C09147=1195.626,20.298,-44.972,-179.612,5.706,148.893
C09148=1195.622,20.548,-44.987,-179.609,5.707,148.893
C09149=1195.617,20.797,-45.002,-179.606,5.707,148.892
C09150=1195.611,21.047,-45.017,-179.604,5.708,148.892
C09151=1195.606,21.296,-45.031,-179.602,5.709,148.891
C09152=1195.602,21.545,-45.046,-179.599,5.709,148.890
C09153=1195.596,21.795,-45.061,-179.596,5.710,148.889
C09154=1195.591,22.045,-45.076,-179.594,5.710,148.889
C09155=1195.586,22.294,-45.091,-179.592,5.711,148.888
C09156=1195.581,22.544,-45.106,-179.589,5.711,148.888
C09157=1195.576,22.793,-45.120,-179.586,5.712,148.887
C09158=1195.571,23.042,-45.135,-179.584,5.713,148.887
C09159=1195.566,23.292,-45.150,-179.581,5.713,148.886
C09160=1195.561,23.542,-45.165,-179.579,5.714,148.885
C09161=1195.556,23.791,-45.180,-179.576,5.714,148.885
C09162=1195.551,24.041,-45.195,-179.574,5.715,148.884
C09163=1195.546,24.290,-45.209,-179.571,5.716,148.883
C09164=1195.541,24.539,-45.224,-179.569,5.716,148.883
C09165=1195.536,24.789,-45.240,-179.566,5.717,148.882
C09166=1195.531,25.039,-45.254,-179.563,5.717,148.881
C09167=1195.526,25.288,-45.269,-179.561,5.718,148.881
C09168=1195.520,25.538,-45.284,-179.558,5.719,148.880
C09169=1195.516,25.787,-45.299,-179.555,5.720,148.880
C09170=1195.510,26.036,-45.315,-179.553,5.720,148.879
C09171=1195.505,26.286,-45.329,-179.551,5.721,148.878
C09172=1195.501,26.536,-45.344,-179.548,5.722,148.878
C09173=1195.496,26.785,-45.360,-179.545,5.722,148.877
C09174=1195.491,27.035,-45.374,-179.543,5.723,148.876
C09175=1195.486,27.284,-45.390,-179.540,5.724,148.876
C09176=1195.481,27.533,-45.405,-179.538,5.724,148.875
C09177=1195.475,27.783,-45.420,-179.535,5.725,148.875
C09178=1195.471,28.032,-45.435,-179.533,5.725,148.874
C09179=1195.465,28.282,-45.450,-179.530,5.726,148.873
C09180=1195.460,28.551,-45.466,-179.528,5.727,148.873
C09181=1195.454,28.820,-45.482,-179.525,5.727,148.872
C09182=1195.449,29.088,-45.499,-179.522,5.728,148.871
C09183=1195.444,29.357,-45.515,-179.519,5.729,148.871
C09184=1195.439,29.606,-45.530,-179.517,5.730,148.870
C09185=1195.434,29.856,-45.546,-179.514,5.730,148.869
C09186=1195.429,30.106,-45.560,-179.512,5.731,148.869
C09187=1195.424,30.355,-45.576,-179.509,5.731,148.868
C09188=1195.419,30.604,-45.591,-179.506,5.732,148.868
C09189=1195.414,30.854,-45.606,-179.504,5.732,148.867
C09190=1195.409,31.104,-45.621,-179.502,5.733,148.866
C09191=1195.403,31.353,-45.636,-179.499,5.734,148.866
C09192=1195.399,31.603,-45.652,-179.496,5.734,148.865
C09193=1195.394,31.852,-45.667,-179.494,5.735,148.865
C09194=1195.389,32.102,-45.683,-179.492,5.736,148.864
C09195=1195.384,32.351,-45.698,-179.489,5.736,148.863
C09196=1195.378,32.601,-45.713,-179.486,5.737,148.863
C09197=1195.374,32.850,-45.728,-179.484,5.738,148.862
C09198=1195.369,33.100,-45.744,-179.481,5.738,148.861
C09199=1195.364,33.349,-45.759,-179.479,5.739,148.861
C09200=1195.359,33.598,-45.774,-179.476,5.740,148.860
C09201=1195.353,33.848,-45.790,-179.473,5.741,148.860
C09202=1195.349,34.097,-45.805,-179.471,5.741,148.859
C09203=1195.344,34.347,-45.821,-179.468,5.742,148.858
C09204=1195.339,34.596,-45.836,-179.466,5.742,148.858
C09205=1195.334,34.845,-45.851,-179.463,5.743,148.857
C09206=1195.328,35.095,-45.866,-179.461,5.744,148.857
C09207=1195.324,35.345,-45.881,-179.458,5.744,148.856
C09208=1195.319,35.595,-45.897,-179.456,5.745,148.855
C09209=1195.313,35.844,-45.913,-179.453,5.746,148.855
C09210=1195.309,36.093,-45.928,-179.451,5.746,148.854
C09211=1195.303,36.343,-45.943,-179.448,5.747,148.853
C09212=1195.299,36.592,-45.959,-179.446,5.748,148.853
C09213=1195.294,36.842,-45.974,-179.443,5.748,148.852
C09214=1195.289,37.091,-45.990,-179.440,5.750,148.852
C09215=1195.283,37.341,-46.005,-179.437,5.750,148.851
C09216=1195.279,37.590,-46.021,-179.435,5.751,148.850
C09217=1195.274,37.840,-46.036,-179.433,5.751,148.850
C09218=1195.268,38.089,-46.052,-179.430,5.752,148.849
C09219=1195.264,38.338,-46.067,-179.428,5.753,148.849
C09220=1195.259,38.588,-46.083,-179.425,5.753,148.848
C09221=1195.254,38.837,-46.099,-179.422,5.754,148.847
C09222=1195.249,39.086,-46.114,-179.420,5.754,148.847
C09223=1195.244,39.336,-46.130,-179.418,5.755,148.846
C09224=1195.239,39.586,-46.146,-179.415,5.756,148.846
C09225=1195.234,39.835,-46.161,-179.412,5.757,148.845
C09226=1195.229,40.084,-46.176,-179.410,5.758,148.844
C09227=1195.224,40.334,-46.192,-179.407,5.759,148.844
C09228=1195.219,40.584,-46.208,-179.404,5.759,148.843
C09229=1195.213,40.833,-46.223,-179.402,5.760,148.842
C09230=1195.209,41.083,-46.239,-179.400,5.761,148.842
C09231=1195.204,41.332,-46.255,-179.397,5.761,148.841
C09232=1195.199,41.581,-46.271,-179.394,5.762,148.841
C09233=1195.194,41.830,-46.286,-179.392,5.762,148.840
C09234=1195.189,42.081,-46.302,-179.389,5.763,148.839
C09235=1195.184,42.330,-46.317,-179.386,5.764,148.839
C09236=1195.179,42.578,-46.334,-179.384,5.765,148.838
C09237=1195.174,42.829,-46.349,-179.381,5.766,148.838
C09238=1195.169,43.078,-46.365,-179.379,5.766,148.837
C09239=1195.163,43.327,-46.381,-179.376,5.767,148.836
C09240=1195.159,43.577,-46.397,-179.374,5.768,148.836
C09241=1195.154,43.826,-46.412,-179.371,5.768,148.835
C09242=1195.150,44.076,-46.428,-179.369,5.769,148.835
C09243=1195.144,44.325,-46.444,-179.366,5.770,148.834
C09244=1195.139,44.575,-46.459,-179.363,5.771,148.833
C09245=1195.134,44.824,-46.476,-179.361,5.771,148.833
C09246=1195.129,45.074,-46.492,-179.358,5.772,148.832
C09247=1195.124,45.323,-46.507,-179.356,5.773,148.832
C09248=1195.120,45.572,-46.523,-179.353,5.773,148.831
C09249=1195.114,45.822,-46.539,-179.351,5.774,148.830
C09250=1195.110,46.072,-46.555,-179.349,5.775,148.830
C09251=1195.105,46.321,-46.571,-179.345,5.776,148.829
C09252=1195.099,46.570,-46.587,-179.343,5.777,148.829
C09253=1195.094,46.820,-46.603,-179.341,5.778,148.828
C09254=1195.089,47.069,-46.619,-179.338,5.778,148.827
C09255=1195.084,47.319,-46.635,-179.335,5.779,148.827
C09256=1195.079,47.568,-46.651,-179.333,5.779,148.826
C09257=1195.074,47.817,-46.667,-179.330,5.780,148.826
C09258=1195.069,48.067,-46.683,-179.327,5.781,148.825
C09259=1195.065,48.316,-46.698,-179.325,5.782,148.824
C09260=1195.060,48.566,-46.715,-179.322,5.783,148.824
C09261=1195.055,48.815,-46.730,-179.320,5.783,148.823
C09262=1195.050,49.065,-46.747,-179.317,5.784,148.823
C09263=1195.045,49.314,-46.762,-179.315,5.785,148.822
C09264=1195.040,49.563,-46.779,-179.312,5.785,148.821
C09265=1195.035,49.813,-46.795,-179.309,5.787,148.821
C09266=1195.030,50.062,-46.811,-179.307,5.787,148.820
C09267=1195.025,50.312,-46.827,-179.304,5.788,148.820
C09268=1195.020,50.561,-46.842,-179.302,5.789,148.819
C09269=1195.015,50.811,-46.859,-179.299,5.789,148.818
C09270=1195.010,51.060,-46.875,-179.297,5.790,148.818
C09271=1195.005,51.310,-46.891,-179.294,5.790,148.817
C09272=1195.000,51.559,-46.907,-179.291,5.792,148.817
C09273=1194.996,51.809,-46.924,-179.289,5.793,148.816
C09274=1194.990,52.057,-46.940,-179.286,5.793,148.815
C09275=1194.986,52.307,-46.956,-179.284,5.794,148.815
C09276=1194.981,52.556,-46.972,-179.282,5.795,148.814
C09277=1194.976,52.806,-46.988,-179.279,5.795,148.814
C09278=1194.971,53.055,-47.004,-179.276,5.797,148.813
C09279=1194.965,53.306,-47.021,-179.274,5.797,148.813
C09280=1194.960,53.554,-47.037,-179.271,5.798,148.812
C09281=1194.955,53.804,-47.053,-179.268,5.799,148.811
C09282=1194.950,54.053,-47.070,-179.266,5.799,148.811
C09283=1194.946,54.303,-47.086,-179.263,5.800,148.810
C09284=1194.940,54.571,-47.103,-179.260,5.801,148.809
C09285=1194.935,54.839,-47.121,-179.258,5.802,148.809
C09286=1194.930,55.108,-47.138,-179.254,5.803,148.808
C09287=1194.924,55.377,-47.156,-179.252,5.804,148.808
C09288=1194.919,55.626,-47.173,-179.250,5.805,148.807
C09289=1194.914,55.875,-47.189,-179.247,5.805,148.806
C09290=1194.909,56.125,-47.205,-179.245,5.806,148.806
C09291=1194.904,56.374,-47.221,-179.242,5.807,148.805
C09292=1194.900,56.624,-47.238,-179.239,5.808,148.805
C09293=1194.894,56.873,-47.253,-179.237,5.809,148.804
C09294=1194.889,57.123,-47.271,-179.234,5.809,148.803
C09295=1194.885,57.372,-47.287,-179.232,5.810,148.803
C09296=1194.880,57.621,-47.304,-179.229,5.812,148.802
C09297=1194.875,57.871,-47.320,-179.226,5.812,148.802
C09298=1194.870,58.120,-47.336,-179.224,5.813,148.801
C09299=1194.865,58.370,-47.353,-179.221,5.814,148.801
C09300=1194.859,58.619,-47.370,-179.219,5.814,148.800
C09301=1194.855,58.869,-47.385,-179.216,5.815,148.799
C09302=1194.850,59.118,-47.402,-179.213,5.816,148.799
C09303=1194.845,59.367,-47.418,-179.211,5.817,148.798
C09304=1194.840,59.617,-47.436,-179.208,5.817,148.798
C09305=1194.835,59.866,-47.452,-179.206,5.818,148.797
C09306=1194.830,60.116,-47.468,-179.203,5.820,148.796
C09307=1194.826,60.365,-47.485,-179.200,5.820,148.796
C09308=1194.820,60.614,-47.502,-179.198,5.821,148.795
C09309=1194.815,60.864,-47.518,-179.195,5.822,148.795
C09310=1194.811,61.113,-47.535,-179.193,5.822,148.794
C09311=1194.806,61.362,-47.551,-179.190,5.824,148.794
C09312=1194.800,61.612,-47.568,-179.187,5.824,148.793
C09313=1194.796,61.862,-47.584,-179.185,5.825,148.792
C09314=1194.791,62.111,-47.601,-179.183,5.826,148.792
C09315=1194.785,62.360,-47.618,-179.179,5.827,148.791
C09316=1194.781,62.610,-47.635,-179.177,5.828,148.791
C09317=1194.776,62.859,-47.651,-179.175,5.829,148.790
C09318=1194.771,63.108,-47.668,-179.172,5.829,148.789
C09319=1194.766,63.358,-47.685,-179.170,5.830,148.789
C09320=1194.761,63.607,-47.701,-179.167,5.831,148.788
C09321=1194.757,63.856,-47.718,-179.164,5.832,148.788
C09322=1194.751,64.106,-47.735,-179.162,5.833,148.787
C09323=1194.746,64.355,-47.751,-179.159,5.833,148.787
C09324=1194.742,64.604,-47.768,-179.157,5.835,148.786
C09325=1194.737,64.854,-47.785,-179.154,5.836,148.785
C09326=1194.731,65.103,-47.802,-179.151,5.836,148.785
C09327=1194.726,65.353,-47.819,-179.149,5.837,148.784
C09328=1194.722,65.602,-47.836,-179.146,5.838,148.784
C09329=1194.717,65.851,-47.852,-179.143,5.839,148.783
C09330=1194.711,66.101,-47.869,-179.141,5.840,148.783
C09331=1194.707,66.350,-47.886,-179.138,5.840,148.782
C09332=1194.703,66.600,-47.902,-179.135,5.842,148.781
C09333=1194.697,66.849,-47.919,-179.133,5.843,148.781
C09334=1194.692,67.098,-47.936,-179.131,5.843,148.780
C09335=1194.687,67.348,-47.953,-179.128,5.844,148.780
C09336=1194.683,67.598,-47.970,-179.125,5.846,148.779
C09337=1194.677,67.847,-47.987,-179.123,5.846,148.778
C09338=1194.672,68.096,-48.004,-179.120,5.847,148.778
C09339=1194.668,68.346,-48.020,-179.118,5.848,148.777
C09340=1194.663,68.595,-48.038,-179.115,5.849,148.777
C09341=1194.658,68.844,-48.055,-179.112,5.850,148.776
C09342=1194.653,69.093,-48.072,-179.110,5.850,148.776
C09343=1194.648,69.343,-48.088,-179.108,5.851,148.775
C09344=1194.643,69.593,-48.106,-179.104,5.853,148.774
C09345=1194.638,69.841,-48.122,-179.102,5.853,148.774
C09346=1194.633,70.091,-48.140,-179.100,5.854,148.773
C09347=1194.628,70.340,-48.157,-179.097,5.855,148.773
C09348=1194.623,70.590,-48.174,-179.094,5.856,148.772
C09349=1194.619,70.839,-48.191,-179.092,5.857,148.772
C09350=1194.613,71.088,-48.207,-179.089,5.857,148.771
C09351=1194.609,71.337,-48.225,-179.087,5.858,148.771
C09352=1194.603,71.587,-48.242,-179.084,5.860,148.770
C09353=1194.599,71.837,-48.259,-179.082,5.861,148.769
C09354=1194.594,72.086,-48.276,-179.079,5.861,148.769
C09355=1194.589,72.335,-48.293,-179.076,5.862,148.768
C09356=1194.584,72.584,-48.310,-179.074,5.863,148.768
C09357=1194.579,72.834,-48.328,-179.071,5.864,148.767
C09358=1194.574,73.084,-48.344,-179.069,5.865,148.767
C09359=1194.569,73.333,-48.362,-179.066,5.866,148.766
C09360=1194.565,73.582,-48.379,-179.063,5.867,148.765
C09361=1194.559,73.831,-48.396,-179.061,5.868,148.765
C09362=1194.555,74.080,-48.413,-179.058,5.869,148.764
C09363=1194.549,74.330,-48.430,-179.055,5.870,148.764
C09364=1194.544,74.580,-48.448,-179.053,5.870,148.763
C09365=1194.540,74.829,-48.465,-179.050,5.871,148.762
C09366=1194.535,75.079,-48.482,-179.047,5.873,148.762
C09367=1194.530,75.328,-48.499,-179.045,5.873,148.761
C09368=1194.525,75.576,-48.517,-179.043,5.874,148.761
C09369=1194.520,75.826,-48.534,-179.040,5.876,148.760
C09370=1194.515,76.075,-48.551,-179.037,5.876,148.760
C09371=1194.510,76.325,-48.569,-179.035,5.877,148.759
C09372=1194.505,76.575,-48.586,-179.032,5.878,148.759
C09373=1194.501,76.824,-48.603,-179.029,5.879,148.758
C09374=1194.496,77.073,-48.621,-179.027,5.880,148.758
C09375=1194.491,77.323,-48.638,-179.025,5.881,148.757
C09376=1194.486,77.572,-48.655,-179.021,5.882,148.756
C09377=1194.481,77.821,-48.673,-179.019,5.883,148.756
C09378=1194.476,78.070,-48.690,-179.017,5.884,148.755
C09379=1194.471,78.319,-48.707,-179.013,5.885,148.755
C09380=1194.466,78.569,-48.725,-179.011,5.886,148.754
C09381=1194.461,78.818,-48.743,-179.009,5.886,148.754
C09382=1194.456,79.068,-48.760,-179.006,5.888,148.753
C09383=1194.452,79.317,-48.777,-179.003,5.889,148.753
C09384=1194.447,79.567,-48.795,-179.001,5.889,148.752
C09385=1194.442,79.816,-48.813,-178.998,5.891,148.751
C09386=1194.436,80.066,-48.830,-178.995,5.892,148.751
C09387=1194.432,80.314,-48.847,-178.993,5.892,148.750
C09388=1194.427,80.583,-48.866,-178.990,5.894,148.750
C09389=1194.421,80.851,-48.885,-178.987,5.894,148.749
C09390=1194.416,81.120,-48.904,-178.984,5.896,148.748
C09391=1194.411,81.388,-48.923,-178.982,5.897,148.748
C09392=1194.406,81.638,-48.940,-178.979,5.898,148.747
C09393=1194.401,81.887,-48.958,-178.977,5.899,148.747
C09394=1194.396,82.136,-48.975,-178.974,5.899,148.746
C09395=1194.391,82.386,-48.993,-178.971,5.901,148.746
C09396=1194.386,82.635,-49.011,-178.969,5.902,148.745
C09397=1194.381,82.885,-49.028,-178.966,5.902,148.745
C09398=1194.377,83.133,-49.046,-178.963,5.904,148.744
C09399=1194.372,83.383,-49.064,-178.961,5.905,148.743
C09400=1194.367,83.632,-49.081,-178.959,5.906,148.743
C09401=1194.362,83.882,-49.099,-178.955,5.907,148.742
C09402=1194.357,84.131,-49.117,-178.953,5.908,148.742
C09403=1194.352,84.380,-49.135,-178.951,5.908,148.741
C09404=1194.347,84.630,-49.152,-178.948,5.910,148.741
C09405=1194.343,84.879,-49.169,-178.945,5.911,148.740
C09406=1194.338,85.128,-49.187,-178.943,5.911,148.740
C09407=1194.333,85.378,-49.205,-178.940,5.913,148.739
C09408=1194.328,85.627,-49.223,-178.937,5.914,148.739
C09409=1194.323,85.876,-49.241,-178.935,5.914,148.738
C09410=1194.318,86.125,-49.259,-178.932,5.916,148.737
C09411=1194.313,86.374,-49.277,-178.930,5.917,148.737
C09412=1194.308,86.624,-49.294,-178.927,5.918,148.736
C09413=1194.303,86.873,-49.312,-178.925,5.919,148.736
C09414=1194.299,87.122,-49.329,-178.922,5.920,148.735
C09415=1194.294,87.371,-49.347,-178.919,5.921,148.735
C09416=1194.289,87.621,-49.366,-178.917,5.922,148.734
C09417=1194.284,87.871,-49.383,-178.914,5.922,148.734
C09418=1194.279,88.120,-49.401,-178.911,5.924,148.733
C09419=1194.274,88.369,-49.419,-178.909,5.925,148.733
C09420=1194.269,88.619,-49.437,-178.906,5.926,148.732
C09421=1194.265,88.868,-49.455,-178.903,5.927,148.731
C09422=1194.260,89.117,-49.473,-178.901,5.928,148.731
C09423=1194.255,89.366,-49.491,-178.898,5.929,148.730
C09424=1194.250,89.615,-49.509,-178.896,5.930,148.730
C09425=1194.245,89.864,-49.527,-178.893,5.931,148.729
C09426=1194.240,90.115,-49.544,-178.891,5.933,148.729
C09427=1194.235,90.364,-49.562,-178.888,5.933,148.728
C09428=1194.230,90.613,-49.580,-178.885,5.935,148.728
C09429=1194.226,90.862,-49.598,-178.883,5.935,148.727
C09430=1194.221,91.112,-49.616,-178.880,5.936,148.727
C09431=1194.216,91.361,-49.634,-178.877,5.938,148.726
C09432=1194.211,91.610,-49.652,-178.875,5.939,148.726
C09433=1194.206,91.859,-49.670,-178.872,5.940,148.725
C09434=1194.202,92.109,-49.688,-178.870,5.941,148.725
C09435=1194.196,92.358,-49.707,-178.867,5.941,148.724
C09436=1194.191,92.608,-49.725,-178.864,5.943,148.723
C09437=1194.186,92.857,-49.743,-178.862,5.944,148.723
C09438=1194.181,93.106,-49.761,-178.859,5.945,148.722
C09439=1194.176,93.355,-49.779,-178.857,5.946,148.722
C09440=1194.172,93.605,-49.797,-178.854,5.947,148.721
C09441=1194.167,93.854,-49.815,-178.851,5.948,148.721
C09442=1194.162,94.103,-49.834,-178.849,5.949,148.720
C09443=1194.158,94.352,-49.852,-178.846,5.951,148.720
C09444=1194.153,94.601,-49.870,-178.843,5.951,148.719
C09445=1194.148,94.851,-49.889,-178.841,5.952,148.719
C09446=1194.143,95.100,-49.907,-178.838,5.954,148.718
C09447=1194.138,95.350,-49.925,-178.836,5.954,148.718
C09448=1194.133,95.599,-49.943,-178.833,5.956,148.717
C09449=1194.128,95.848,-49.961,-178.830,5.957,148.717
C09450=1194.124,96.098,-49.979,-178.827,5.958,148.716
C09451=1194.119,96.346,-49.998,-178.825,5.959,148.715
C09452=1194.113,96.596,-50.016,-178.822,5.960,148.715
C09453=1194.108,96.845,-50.034,-178.820,5.961,148.714
C09454=1194.104,97.095,-50.053,-178.817,5.962,148.714
C09455=1194.099,97.344,-50.071,-178.814,5.964,148.713
C09456=1194.095,97.593,-50.089,-178.812,5.965,148.713
C09457=1194.089,97.842,-50.108,-178.810,5.965,148.712
C09458=1194.084,98.091,-50.126,-178.807,5.967,148.712
C09459=1194.080,98.341,-50.144,-178.804,5.967,148.711
C09460=1194.075,98.590,-50.163,-178.802,5.969,148.711
C09461=1194.069,98.839,-50.182,-178.799,5.970,148.710
C09462=1194.065,99.089,-50.200,-178.796,5.972,148.710
C09463=1194.060,99.338,-50.218,-178.794,5.972,148.709
C09464=1194.056,99.587,-50.237,-178.791,5.974,148.709
C09465=1194.050,99.836,-50.255,-178.788,5.974,148.708
C09466=1194.046,100.086,-50.274,-178.786,5.975,148.708
C09467=1194.041,100.335,-50.292,-178.783,5.977,148.707
C09468=1194.036,100.584,-50.310,-178.781,5.978,148.707
C09469=1194.031,100.834,-50.329,-178.778,5.979,148.706
C09470=1194.026,101.083,-50.348,-178.776,5.980,148.706
C09471=1194.022,101.332,-50.366,-178.772,5.981,148.705
C09472=1194.016,101.581,-50.384,-178.770,5.982,148.704
C09473=1194.012,101.831,-50.403,-178.767,5.984,148.704
C09474=1194.007,102.080,-50.421,-178.765,5.985,148.703
C09475=1194.001,102.329,-50.440,-178.762,5.986,148.703
C09476=1193.997,102.579,-50.459,-178.760,5.987,148.702
C09477=1193.992,102.828,-50.477,-178.758,5.988,148.702
C09478=1193.987,103.077,-50.496,-178.754,5.989,148.701
C09479=1193.983,103.327,-50.515,-178.752,5.990,148.701
C09480=1193.978,103.575,-50.533,-178.749,5.992,148.700
C09481=1193.973,103.825,-50.552,-178.747,5.992,148.700
C09482=1193.968,104.074,-50.570,-178.744,5.994,148.699
C09483=1193.964,104.323,-50.589,-178.742,5.995,148.699
C09484=1193.959,104.573,-50.608,-178.738,5.996,148.698
C09485=1193.954,104.822,-50.627,-178.736,5.997,148.698
C09486=1193.948,105.071,-50.645,-178.733,5.998,148.697
C09487=1193.944,105.320,-50.664,-178.731,5.999,148.697
C09488=1193.939,105.570,-50.682,-178.728,6.001,148.696
C09489=1193.934,105.819,-50.702,-178.726,6.002,148.696
C09490=1193.930,106.068,-50.721,-178.723,6.003,148.695
C09491=1193.924,106.317,-50.739,-178.720,6.004,148.695
C09492=1193.920,106.586,-50.760,-178.718,6.006,148.694
C09493=1193.914,106.854,-50.780,-178.715,6.006,148.694
C09494=1193.909,107.123,-50.800,-178.712,6.008,148.693
C09495=1193.904,107.391,-50.820,-178.709,6.009,148.693
C09496=1193.899,107.640,-50.839,-178.706,6.010,148.692
C09497=1193.894,107.889,-50.857,-178.704,6.012,148.691
C09498=1193.889,108.139,-50.877,-178.701,6.012,148.691
C09499=1193.884,108.388,-50.895,-178.698,6.014,148.690
C09500=1193.880,108.637,-50.915,-178.696,6.015,148.690
C09501=1193.875,108.886,-50.933,-178.693,6.016,148.689
C09502=1193.870,109.136,-50.952,-178.691,6.017,148.689
C09503=1193.865,109.385,-50.971,-178.688,6.019,148.688
C09504=1193.861,109.634,-50.991,-178.686,6.020,148.688
C09505=1193.856,109.883,-51.009,-178.682,6.021,148.687
C09506=1193.850,110.132,-51.028,-178.680,6.022,148.687
C09507=1193.846,110.382,-51.047,-178.678,6.024,148.686
C09508=1193.841,110.631,-51.066,-178.675,6.024,148.686
C09509=1193.836,110.881,-51.085,-178.672,6.026,148.685
C09510=1193.831,111.129,-51.104,-178.670,6.027,148.685
C09511=1193.827,111.379,-51.124,-178.667,6.028,148.684
C09512=1193.822,111.628,-51.142,-178.665,6.029,148.684
C09513=1193.817,111.878,-51.161,-178.662,6.031,148.683
C09514=1193.812,112.126,-51.180,-178.660,6.032,148.683
C09515=1193.808,112.376,-51.200,-178.656,6.033,148.682
C09516=1193.802,112.625,-51.219,-178.654,6.034,148.682
C09517=1193.798,112.874,-51.237,-178.651,6.035,148.681
C09518=1193.793,113.123,-51.257,-178.648,6.037,148.681
C09519=1193.788,113.373,-51.276,-178.646,6.038,148.680
C09520=1193.783,113.621,-51.295,-178.643,6.040,148.680
C09521=1193.779,113.871,-51.315,-178.641,6.040,148.679
C09522=1193.774,114.119,-51.333,-178.638,6.042,148.679
C09523=1193.769,114.370,-51.352,-178.636,6.043,148.678
C09524=1193.764,114.619,-51.371,-178.633,6.045,148.678
C09525=1193.760,114.868,-51.391,-178.630,6.045,148.677
C09526=1193.754,115.117,-51.410,-178.628,6.047,148.677
C09527=1193.750,115.366,-51.429,-178.625,6.047,148.676
C09528=1193.745,115.616,-51.449,-178.622,6.049,148.676
C09529=1193.740,115.864,-51.468,-178.620,6.050,148.675
C09530=1193.735,116.114,-51.488,-178.617,6.052,148.675
C09531=1193.730,116.363,-51.507,-178.614,6.053,148.674
C09532=1193.726,116.612,-51.526,-178.612,6.054,148.674
C09533=1193.721,116.861,-51.545,-178.609,6.056,148.673
C09534=1193.716,117.110,-51.565,-178.607,6.057,148.673
C09535=1193.711,117.360,-51.584,-178.604,6.058,148.672
C09536=1193.707,117.609,-51.603,-178.602,6.059,148.672
C09537=1193.702,117.858,-51.623,-178.599,6.061,148.672
C09538=1193.697,118.107,-51.642,-178.596,6.061,148.671
C09539=1193.692,118.357,-51.662,-178.594,6.063,148.671
C09540=1193.688,118.606,-51.681,-178.590,6.064,148.670
C09541=1193.683,118.855,-51.700,-178.588,6.065,148.669
C09542=1193.678,119.104,-51.720,-178.586,6.067,148.669
C09543=1193.672,119.353,-51.739,-178.583,6.068,148.668
C09544=1193.668,119.603,-51.759,-178.580,6.069,148.668
C09545=1193.664,119.852,-51.778,-178.578,6.070,148.668
C09546=1193.658,120.101,-51.797,-178.575,6.072,148.667
C09547=1193.654,120.350,-51.817,-178.573,6.073,148.667
C09548=1193.649,120.600,-51.836,-178.570,6.074,148.666
C09549=1193.643,120.849,-51.856,-178.567,6.076,148.666
C09550=1193.639,121.098,-51.875,-178.565,6.077,148.665
C09551=1193.634,121.346,-51.895,-178.562,6.078,148.665
C09552=1193.630,121.596,-51.914,-178.559,6.079,148.664
C09553=1193.625,121.846,-51.934,-178.557,6.081,148.664
C09554=1193.620,122.094,-51.953,-178.554,6.082,148.663
C09555=1193.615,122.344,-51.973,-178.551,6.083,148.663
C09556=1193.610,122.594,-51.993,-178.549,6.085,148.662
C09557=1193.606,122.841,-52.012,-178.546,6.086,148.662
C09558=1193.601,123.091,-52.032,-178.543,6.087,148.661
C09559=1193.596,123.341,-52.051,-178.541,6.088,148.661
C09560=1193.592,123.590,-52.071,-178.538,6.090,148.660
C09561=1193.587,123.838,-52.091,-178.535,6.091,148.660
C09562=1193.582,124.088,-52.111,-178.533,6.092,148.659
C09563=1193.577,124.338,-52.130,-178.530,6.094,148.659
C09564=1193.572,124.586,-52.150,-178.528,6.095,148.658
C09565=1193.567,124.835,-52.170,-178.525,6.096,148.658
C09566=1193.563,125.085,-52.190,-178.522,6.098,148.657
C09567=1193.558,125.335,-52.209,-178.520,6.099,148.657
C09568=1193.553,125.583,-52.229,-178.517,6.101,148.657
C09569=1193.548,125.832,-52.249,-178.515,6.101,148.656
C09570=1193.543,126.082,-52.269,-178.512,6.103,148.656
C09571=1193.539,126.331,-52.289,-178.509,6.105,148.655
C09572=1193.534,126.580,-52.308,-178.507,6.105,148.655
C09573=1193.529,126.829,-52.328,-178.504,6.107,148.654
C09574=1193.524,127.078,-52.348,-178.501,6.109,148.654
C09575=1193.520,127.328,-52.368,-178.499,6.109,148.653
C09576=1193.514,127.577,-52.387,-178.496,6.111,148.653
C09577=1193.510,127.826,-52.408,-178.494,6.112,148.652
C09578=1193.505,128.075,-52.427,-178.491,6.114,148.652
C09579=1193.501,128.324,-52.448,-178.488,6.115,148.651
C09580=1193.495,128.573,-52.467,-178.486,6.116,148.651
C09581=1193.491,128.822,-52.487,-178.483,6.118,148.650
C09582=1193.486,129.072,-52.507,-178.480,6.119,148.650
C09583=1193.482,129.320,-52.527,-178.478,6.120,148.650
C09584=1193.477,129.570,-52.547,-178.475,6.122,148.649
C09585=1193.472,129.819,-52.566,-178.473,6.123,148.648
C09586=1193.467,130.068,-52.587,-178.470,6.124,148.648
C09587=1193.462,130.317,-52.606,-178.467,6.126,148.647
C09588=1193.458,130.566,-52.627,-178.465,6.127,148.647
C09589=1193.453,130.816,-52.646,-178.462,6.129,148.647
C09590=1193.448,131.064,-52.666,-178.459,6.130,148.646
C09591=1193.443,131.313,-52.687,-178.457,6.131,148.646
C09592=1193.438,131.563,-52.707,-178.454,6.133,148.645
C09593=1193.434,131.812,-52.727,-178.451,6.134,148.645
C09594=1193.429,132.062,-52.747,-178.449,6.135,148.644
C09595=1193.425,132.310,-52.767,-178.446,6.137,148.644
C09596=1193.419,132.579,-52.789,-178.443,6.139,148.643
C09597=1193.414,132.847,-52.811,-178.440,6.140,148.643
C09598=1193.409,133.116,-52.833,-178.438,6.141,148.642
C09599=1193.404,133.385,-52.854,-178.435,6.142,148.642
C09600=1193.399,133.634,-52.874,-178.432,6.144,148.641
C09601=1193.394,133.883,-52.895,-178.429,6.146,148.641
C09602=1193.389,134.133,-52.915,-178.427,6.146,148.640
C09603=1193.384,134.381,-52.935,-178.424,6.148,148.640
C09604=1193.380,134.630,-52.955,-178.422,6.150,148.640
C09605=1193.375,134.880,-52.975,-178.419,6.151,148.639
C09606=1193.370,135.129,-52.996,-178.416,6.152,148.639
C09607=1193.366,135.378,-53.016,-178.414,6.154,148.638
C09608=1193.361,135.627,-53.036,-178.411,6.155,148.638
C09609=1193.356,135.876,-53.056,-178.408,6.156,148.637
C09610=1193.351,136.126,-53.077,-178.406,6.158,148.637
C09611=1193.347,136.375,-53.097,-178.403,6.159,148.636
C09612=1193.342,136.624,-53.118,-178.400,6.161,148.636
C09613=1193.336,136.873,-53.138,-178.398,6.162,148.635
C09614=1193.332,137.122,-53.158,-178.395,6.163,148.635
C09615=1193.327,137.371,-53.178,-178.393,6.165,148.635
C09616=1193.323,137.620,-53.199,-178.390,6.167,148.634
C09617=1193.318,137.869,-53.220,-178.387,6.167,148.634
C09618=1193.313,138.118,-53.239,-178.385,6.169,148.633
C09619=1193.309,138.367,-53.260,-178.382,6.171,148.633
C09620=1193.303,138.617,-53.281,-178.380,6.172,148.632
C09621=1193.299,138.866,-53.301,-178.377,6.173,148.632
C09622=1193.295,139.114,-53.321,-178.374,6.175,148.632
C09623=1193.289,139.364,-53.342,-178.371,6.177,148.631
C09624=1193.285,139.613,-53.362,-178.369,6.178,148.630
C09625=1193.280,139.862,-53.382,-178.366,6.179,148.630
C09626=1193.275,140.112,-53.403,-178.363,6.181,148.630
C09627=1193.271,140.360,-53.424,-178.361,6.182,148.629
C09628=1193.266,140.609,-53.444,-178.358,6.183,148.629
C09629=1193.261,140.859,-53.465,-178.355,6.185,148.628
C09630=1193.257,141.108,-53.486,-178.353,6.186,148.628
C09631=1193.251,141.357,-53.506,-178.351,6.188,148.628
C09632=1193.247,141.606,-53.527,-178.348,6.189,148.627
C09633=1193.243,141.855,-53.547,-178.345,6.191,148.627
C09634=1193.237,142.104,-53.568,-178.343,6.192,148.626
C09635=1193.233,142.353,-53.589,-178.340,6.194,148.626
C09636=1193.228,142.602,-53.610,-178.337,6.195,148.625
C09637=1193.223,142.851,-53.630,-178.335,6.196,148.625
C09638=1193.218,143.100,-53.651,-178.332,6.198,148.624
C09639=1193.214,143.349,-53.671,-178.329,6.200,148.624
C09640=1193.209,143.599,-53.692,-178.327,6.202,148.624
C09641=1193.204,143.848,-53.713,-178.324,6.202,148.623
C09642=1193.200,144.097,-53.733,-178.321,6.204,148.623
C09643=1193.194,144.346,-53.754,-178.319,6.206,148.622
C09644=1193.191,144.595,-53.775,-178.316,6.207,148.622
C09645=1193.185,144.845,-53.796,-178.313,6.208,148.621
C09646=1193.181,145.093,-53.817,-178.311,6.210,148.621
C09647=1193.176,145.342,-53.838,-178.308,6.212,148.620
C09648=1193.172,145.591,-53.858,-178.305,6.213,148.620
C09649=1193.167,145.841,-53.879,-178.303,6.214,148.620
C09650=1193.161,146.090,-53.900,-178.300,6.216,148.619
C09651=1193.157,146.339,-53.920,-178.297,6.218,148.619
C09652=1193.152,146.588,-53.941,-178.295,6.218,148.618
C09653=1193.148,146.836,-53.962,-178.293,6.220,148.618
C09654=1193.142,147.086,-53.983,-178.289,6.222,148.617
C09655=1193.139,147.335,-54.004,-178.287,6.223,148.617
C09656=1193.133,147.584,-54.025,-178.285,6.224,148.617
C09657=1193.129,147.833,-54.045,-178.282,6.226,148.616
C09658=1193.124,148.082,-54.067,-178.279,6.228,148.616
C09659=1193.119,148.331,-54.088,-178.276,6.229,148.615
C09660=1193.115,148.580,-54.108,-178.274,6.230,148.615
C09661=1193.110,148.829,-54.130,-178.271,6.232,148.614
C09662=1193.106,149.079,-54.151,-178.269,6.234,148.614
C09663=1193.101,149.328,-54.172,-178.266,6.236,148.614
C09664=1193.095,149.577,-54.193,-178.263,6.237,148.613
C09665=1193.091,149.825,-54.214,-178.261,6.238,148.613
C09666=1193.086,150.075,-54.235,-178.258,6.240,148.612
C09667=1193.081,150.324,-54.256,-178.255,6.242,148.612
C09668=1193.077,150.573,-54.277,-178.253,6.243,148.612
C09669=1193.072,150.822,-54.298,-178.251,6.244,148.611
C09670=1193.067,151.071,-54.319,-178.247,6.246,148.611
C09671=1193.063,151.320,-54.340,-178.245,6.248,148.610
C09672=1193.058,151.569,-54.361,-178.242,6.249,148.610
C09673=1193.053,151.818,-54.383,-178.240,6.250,148.609
C09674=1193.048,152.068,-54.404,-178.237,6.252,148.609
C09675=1193.044,152.317,-54.425,-178.235,6.254,148.609
C09676=1193.039,152.565,-54.446,-178.231,6.255,148.608
C09677=1193.034,152.815,-54.467,-178.229,6.257,148.608
C09678=1193.030,153.063,-54.488,-178.227,6.258,148.607
C09679=1193.025,153.313,-54.510,-178.224,6.260,148.607
C09680=1193.020,153.561,-54.531,-178.221,6.262,148.606
C09681=1193.015,153.811,-54.552,-178.219,6.263,148.606
C09682=1193.011,154.059,-54.573,-178.215,6.265,148.606
C09683=1193.006,154.309,-54.595,-178.213,6.266,148.605
C09684=1193.002,154.558,-54.616,-178.211,6.267,148.605
C09685=1192.996,154.807,-54.637,-178.208,6.269,148.604
C09686=1192.992,155.056,-54.659,-178.205,6.271,148.604
C09687=1192.988,155.305,-54.680,-178.203,6.273,148.604
C09688=1192.983,155.554,-54.702,-178.200,6.273,148.603
C09689=1192.978,155.803,-54.723,-178.197,6.275,148.603
C09690=1192.973,156.052,-54.744,-178.195,6.277,148.602
C09691=1192.968,156.302,-54.766,-178.192,6.279,148.602
C09692=1192.964,156.550,-54.787,-178.189,6.281,148.602
C09693=1192.959,156.799,-54.808,-178.187,6.281,148.601
C09694=1192.955,157.049,-54.830,-178.184,6.283,148.601
C09695=1192.950,157.297,-54.851,-178.181,6.285,148.600
C09696=1192.945,157.547,-54.872,-178.179,6.286,148.600
C09697=1192.940,157.795,-54.894,-178.176,6.288,148.599
C09698=1192.935,158.045,-54.916,-178.174,6.289,148.599
C09699=1192.930,158.294,-54.937,-178.171,6.291,148.599
C09700=1192.926,158.562,-54.960,-178.168,6.293,148.598
C09701=1192.920,158.832,-54.984,-178.165,6.294,148.598
C09702=1192.916,159.101,-55.007,-178.163,6.296,148.597
C09703=1192.910,159.369,-55.031,-178.159,6.299,148.597
C09704=1192.905,159.619,-55.052,-178.157,6.300,148.597
C09705=1192.902,159.868,-55.073,-178.154,6.301,148.596
C09706=1192.897,160.116,-55.095,-178.151,6.303,148.596
C09707=1192.892,160.365,-55.116,-178.149,6.305,148.595
C09708=1192.887,160.615,-55.138,-178.146,6.306,148.595
C09709=1192.883,160.864,-55.159,-178.143,6.308,148.594
C09710=1192.878,161.112,-55.181,-178.141,6.309,148.594
C09711=1192.873,161.361,-55.203,-178.139,6.311,148.594
C09712=1192.868,161.611,-55.224,-178.136,6.313,148.593
C09713=1192.863,161.859,-55.246,-178.133,6.314,148.593
C09714=1192.859,162.109,-55.268,-178.130,6.316,148.592
C09715=1192.854,162.357,-55.290,-178.127,6.318,148.592
C09716=1192.850,162.607,-55.312,-178.125,6.319,148.592
C09717=1192.845,162.855,-55.333,-178.123,6.320,148.591
C09718=1192.840,163.104,-55.355,-178.120,6.322,148.591
C09719=1192.836,163.354,-55.376,-178.117,6.324,148.591
C09720=1192.831,163.603,-55.398,-178.115,6.326,148.590
C09721=1192.826,163.852,-55.420,-178.112,6.328,148.590
C09722=1192.822,164.101,-55.442,-178.109,6.329,148.589
C09723=1192.817,164.350,-55.464,-178.107,6.330,148.589
C09724=1192.812,164.599,-55.485,-178.104,6.332,148.588
C09725=1192.808,164.847,-55.507,-178.101,6.334,148.588
C09726=1192.803,165.097,-55.530,-178.099,6.335,148.588
C09727=1192.798,165.345,-55.551,-178.096,6.337,148.587
C09728=1192.793,165.595,-55.574,-178.093,6.339,148.587
C09729=1192.789,165.843,-55.595,-178.091,6.341,148.587
C09730=1192.784,166.093,-55.617,-178.088,6.342,148.586
C09731=1192.779,166.341,-55.639,-178.086,6.343,148.586
C09732=1192.775,166.591,-55.661,-178.083,6.345,148.585
C09733=1192.770,166.839,-55.683,-178.080,6.347,148.585
C09734=1192.766,167.089,-55.705,-178.078,6.349,148.585
C09735=1192.760,167.338,-55.727,-178.075,6.350,148.584
C09736=1192.756,167.587,-55.749,-178.072,6.352,148.584
C09737=1192.751,167.836,-55.771,-178.069,6.354,148.583
C09738=1192.747,168.085,-55.793,-178.067,6.356,148.583
C09739=1192.742,168.334,-55.814,-178.065,6.357,148.583
C09740=1192.738,168.583,-55.837,-178.062,6.358,148.582
C09741=1192.733,168.831,-55.859,-178.059,6.360,148.582
C09742=1192.728,169.081,-55.882,-178.056,6.362,148.582
C09743=1192.723,169.329,-55.903,-178.054,6.364,148.581
C09744=1192.719,169.579,-55.925,-178.051,6.365,148.581
C09745=1192.714,169.827,-55.947,-178.048,6.367,148.580
C09746=1192.709,170.077,-55.970,-178.046,6.369,148.580
C09747=1192.705,170.325,-55.992,-178.043,6.371,148.580
C09748=1192.701,170.574,-56.014,-178.040,6.373,148.579
C09749=1192.696,170.823,-56.036,-178.038,6.374,148.579
C09750=1192.691,171.073,-56.058,-178.036,6.375,148.579
C09751=1192.686,171.321,-56.080,-178.033,6.377,148.578
C09752=1192.682,171.570,-56.103,-178.030,6.379,148.578
C09753=1192.676,171.819,-56.125,-178.027,6.380,148.577
C09754=1192.672,172.068,-56.147,-178.025,6.382,148.577
C09755=1192.668,172.318,-56.169,-178.022,6.384,148.577
C09756=1192.663,172.566,-56.192,-178.019,6.386,148.576
C09757=1192.658,172.815,-56.214,-178.016,6.388,148.576
C09758=1192.653,173.064,-56.236,-178.014,6.389,148.575
C09759=1192.649,173.313,-56.259,-178.011,6.391,148.575
C09760=1192.644,173.562,-56.281,-178.008,6.393,148.575
C09761=1192.639,173.811,-56.303,-178.006,6.394,148.574
C09762=1192.635,174.060,-56.326,-178.004,6.396,148.574
C09763=1192.630,174.309,-56.348,-178.001,6.398,148.574
C09764=1192.626,174.558,-56.370,-177.998,6.399,148.573
C09765=1192.622,174.807,-56.393,-177.996,6.401,148.573
C09766=1192.616,175.056,-56.415,-177.993,6.403,148.573
C09767=1192.612,175.305,-56.437,-177.990,6.405,148.572
C09768=1192.606,175.553,-56.460,-177.988,6.406,148.572
C09769=1192.602,175.803,-56.482,-177.985,6.408,148.571
C09770=1192.598,176.051,-56.505,-177.982,6.410,148.571
C09771=1192.593,176.300,-56.527,-177.980,6.412,148.571
C09772=1192.589,176.549,-56.550,-177.977,6.414,148.570
C09773=1192.584,176.799,-56.573,-177.974,6.415,148.570
C09774=1192.579,177.047,-56.595,-177.972,6.417,148.570
C09775=1192.575,177.296,-56.617,-177.969,6.419,148.569
C09776=1192.570,177.545,-56.640,-177.966,6.421,148.569
C09777=1192.565,177.794,-56.662,-177.964,6.423,148.569
C09778=1192.560,178.043,-56.686,-177.962,6.424,148.568
C09779=1192.556,178.292,-56.708,-177.959,6.425,148.568
C09780=1192.551,178.540,-56.731,-177.956,6.427,148.567
C09781=1192.547,178.790,-56.753,-177.954,6.429,148.567
C09782=1192.542,179.039,-56.776,-177.951,6.431,148.567
C09783=1192.537,179.287,-56.798,-177.948,6.433,148.566
C09784=1192.532,179.536,-56.821,-177.946,6.434,148.566
C09785=1192.528,179.785,-56.844,-177.943,6.436,148.566
C09786=1192.523,180.035,-56.866,-177.940,6.438,148.565
C09787=1192.519,180.283,-56.889,-177.938,6.440,148.565
C09788=1192.514,180.533,-56.911,-177.935,6.442,148.565
C09789=1192.510,180.781,-56.934,-177.932,6.443,148.564
C09790=1192.505,181.030,-56.958,-177.930,6.445,148.564
C09791=1192.500,181.279,-56.979,-177.927,6.447,148.564
C09792=1192.496,181.528,-57.003,-177.924,6.449,148.563
C09793=1192.491,181.777,-57.026,-177.922,6.450,148.563
C09794=1192.487,182.026,-57.048,-177.919,6.452,148.562
C09795=1192.481,182.275,-57.071,-177.916,6.454,148.562
C09796=1192.477,182.523,-57.094,-177.914,6.456,148.562
C09797=1192.473,182.772,-57.117,-177.911,6.458,148.561
C09798=1192.468,183.022,-57.139,-177.908,6.459,148.561
C09799=1192.463,183.270,-57.162,-177.906,6.461,148.561
C09800=1192.458,183.519,-57.186,-177.903,6.463,148.560
C09801=1192.454,183.768,-57.208,-177.900,6.465,148.560
C09802=1192.449,184.017,-57.231,-177.898,6.467,148.560
C09803=1192.445,184.267,-57.254,-177.895,6.468,148.559
C09804=1192.440,184.536,-57.279,-177.892,6.470,148.559
C09805=1192.435,184.806,-57.304,-177.890,6.472,148.559
C09806=1192.430,185.075,-57.328,-177.886,6.475,148.558
C09807=1192.425,185.344,-57.354,-177.884,6.476,148.558
C09808=1192.420,185.593,-57.376,-177.881,6.478,148.558
C09809=1192.416,185.842,-57.399,-177.878,6.480,148.557
C09810=1192.411,186.091,-57.422,-177.876,6.482,148.557
C09811=1192.406,186.340,-57.446,-177.873,6.484,148.556
C09812=1192.402,186.589,-57.469,-177.870,6.485,148.556
C09813=1192.398,186.838,-57.492,-177.868,6.487,148.556
C09814=1192.392,187.086,-57.515,-177.865,6.489,148.555
C09815=1192.388,187.335,-57.538,-177.862,6.491,148.555
C09816=1192.383,187.584,-57.562,-177.860,6.493,148.555
C09817=1192.379,187.833,-57.584,-177.857,6.494,148.554
C09818=1192.374,188.082,-57.608,-177.855,6.497,148.554
C09819=1192.370,188.331,-57.631,-177.852,6.498,148.554
C09820=1192.365,188.580,-57.654,-177.849,6.500,148.553
C09821=1192.360,188.828,-57.677,-177.847,6.502,148.553
C09822=1192.356,189.077,-57.700,-177.844,6.504,148.553
C09823=1192.351,189.326,-57.724,-177.842,6.506,148.552
C09824=1192.346,189.575,-57.747,-177.839,6.507,148.552
C09825=1192.342,189.824,-57.770,-177.836,6.509,148.552
C09826=1192.338,190.073,-57.793,-177.834,6.511,148.551
C09827=1192.333,190.322,-57.816,-177.831,6.513,148.551
C09828=1192.328,190.571,-57.840,-177.828,6.515,148.551
C09829=1192.323,190.820,-57.863,-177.826,6.516,148.550
C09830=1192.319,191.069,-57.886,-177.822,6.519,148.550
C09831=1192.313,191.317,-57.909,-177.820,6.521,148.550
C09832=1192.309,191.566,-57.932,-177.817,6.523,148.550
C09833=1192.305,191.815,-57.956,-177.815,6.525,148.549
C09834=1192.300,192.064,-57.980,-177.812,6.527,148.549
C09835=1192.296,192.313,-58.003,-177.809,6.528,148.548
C09836=1192.291,192.562,-58.026,-177.807,6.530,148.548
C09837=1192.286,192.811,-58.050,-177.804,6.532,148.548
C09838=1192.282,193.060,-58.073,-177.801,6.534,148.547
C09839=1192.277,193.309,-58.096,-177.799,6.536,148.547
C09840=1192.272,193.557,-58.120,-177.796,6.537,148.547
C09841=1192.268,193.806,-58.144,-177.794,6.540,148.547
C09842=1192.263,194.055,-58.167,-177.791,6.541,148.546
C09843=1192.258,194.304,-58.191,-177.789,6.543,148.546
C09844=1192.255,194.552,-58.214,-177.786,6.545,148.546
C09845=1192.250,194.801,-58.237,-177.783,6.547,148.545
C09846=1192.245,195.050,-58.261,-177.781,6.549,148.545
C09847=1192.241,195.299,-58.284,-177.777,6.551,148.545
C09848=1192.236,195.548,-58.308,-177.775,6.553,148.544
C09849=1192.232,195.797,-58.332,-177.773,6.555,148.544
C09850=1192.227,196.046,-58.355,-177.770,6.557,148.544
C09851=1192.222,196.294,-58.379,-177.767,6.559,148.543
C09852=1192.218,196.543,-58.402,-177.765,6.561,148.543
C09853=1192.213,196.792,-58.426,-177.762,6.562,148.543
C09854=1192.209,197.041,-58.450,-177.759,6.564,148.542
C09855=1192.204,197.290,-58.473,-177.757,6.566,148.542
C09856=1192.199,197.539,-58.498,-177.754,6.568,148.542
C09857=1192.194,197.788,-58.521,-177.752,6.570,148.541
C09858=1192.189,198.037,-58.545,-177.749,6.572,148.541
C09859=1192.185,198.285,-58.569,-177.746,6.574,148.541
C09860=1192.180,198.534,-58.592,-177.743,6.576,148.540
C09861=1192.176,198.782,-58.616,-177.741,6.578,148.540
C09862=1192.172,199.032,-58.640,-177.738,6.580,148.540
C09863=1192.167,199.281,-58.664,-177.735,6.582,148.539
C09864=1192.163,199.530,-58.687,-177.733,6.584,148.539
C09865=1192.158,199.778,-58.711,-177.730,6.585,148.539
C09866=1192.154,200.027,-58.735,-177.728,6.587,148.539
C09867=1192.149,200.275,-58.759,-177.725,6.589,148.538
C09868=1192.144,200.525,-58.783,-177.722,6.591,148.538
C09869=1192.139,200.773,-58.807,-177.719,6.594,148.538
C09870=1192.135,201.022,-58.830,-177.717,6.595,148.537
C09871=1192.130,201.271,-58.854,-177.714,6.597,148.537
C09872=1192.126,201.520,-58.878,-177.712,6.599,148.537
C09873=1192.122,201.769,-58.902,-177.709,6.601,148.536
C09874=1192.116,202.018,-58.926,-177.706,6.603,148.536
C09875=1192.112,202.267,-58.950,-177.704,6.605,148.536
C09876=1192.108,202.515,-58.974,-177.701,6.607,148.535
C09877=1192.103,202.764,-58.997,-177.698,6.610,148.535
C09878=1192.099,203.012,-59.022,-177.696,6.611,148.535
C09879=1192.094,203.262,-59.047,-177.693,6.613,148.535
C09880=1192.089,203.511,-59.070,-177.690,6.615,148.534
C09881=1192.085,203.759,-59.094,-177.688,6.617,148.534
C09882=1192.081,204.008,-59.118,-177.686,6.619,148.534
C09883=1192.076,204.257,-59.141,-177.683,6.621,148.533
C09884=1192.071,204.505,-59.166,-177.680,6.623,148.533
C09885=1192.067,204.755,-59.191,-177.677,6.625,148.533
C09886=1192.062,205.003,-59.215,-177.674,6.627,148.532
C09887=1192.057,205.252,-59.239,-177.672,6.629,148.532
C09888=1192.053,205.501,-59.263,-177.670,6.631,148.532
C09889=1192.048,205.749,-59.287,-177.667,6.633,148.532
C09890=1192.044,205.998,-59.311,-177.664,6.635,148.531
C09891=1192.039,206.248,-59.335,-177.662,6.636,148.531
C09892=1192.035,206.496,-59.359,-177.658,6.639,148.531
C09893=1192.030,206.744,-59.383,-177.656,6.641,148.531
C09894=1192.025,206.993,-59.408,-177.654,6.643,148.530
C09895=1192.021,207.242,-59.432,-177.651,6.645,148.530
C09896=1192.017,207.491,-59.456,-177.648,6.647,148.530
C09897=1192.011,207.740,-59.480,-177.646,6.648,148.529
C09898=1192.007,207.988,-59.504,-177.643,6.651,148.529
C09899=1192.003,208.238,-59.529,-177.640,6.653,148.529
C09900=1191.998,208.486,-59.554,-177.638,6.655,148.528
C09901=1191.994,208.735,-59.578,-177.635,6.657,148.528
C09902=1191.989,208.983,-59.602,-177.633,6.659,148.528
C09903=1191.985,209.233,-59.627,-177.630,6.661,148.528
C09904=1191.980,209.481,-59.651,-177.627,6.663,148.527
C09905=1191.975,209.730,-59.675,-177.624,6.665,148.527
C09906=1191.971,209.978,-59.700,-177.622,6.667,148.527
C09907=1191.966,210.228,-59.724,-177.619,6.669,148.527
C09908=1191.961,210.498,-59.751,-177.617,6.671,148.526
C09909=1191.957,210.768,-59.777,-177.613,6.674,148.526
C09910=1191.951,211.038,-59.803,-177.611,6.675,148.526
C09911=1191.947,211.309,-59.831,-177.608,6.678,148.525
C09912=1191.942,211.558,-59.855,-177.605,6.680,148.525
C09913=1191.937,211.806,-59.879,-177.602,6.682,148.525
C09914=1191.933,212.056,-59.904,-177.600,6.684,148.524
C09915=1191.928,212.304,-59.928,-177.597,6.686,148.524
C09916=1191.923,212.553,-59.953,-177.594,6.688,148.524
C09917=1191.919,212.802,-59.977,-177.592,6.690,148.523
C09918=1191.914,213.051,-60.002,-177.589,6.692,148.523
C09919=1191.910,213.299,-60.026,-177.587,6.694,148.523
C09920=1191.905,213.549,-60.051,-177.584,6.697,148.523
C09921=1191.901,213.796,-60.076,-177.581,6.699,148.522
C09922=1191.896,214.045,-60.101,-177.579,6.701,148.522
C09923=1191.892,214.294,-60.125,-177.576,6.702,148.522
C09924=1191.887,214.543,-60.150,-177.573,6.704,148.522
C09925=1191.882,214.792,-60.174,-177.570,6.707,148.521
C09926=1191.878,215.041,-60.199,-177.568,6.709,148.521
C09927=1191.873,215.289,-60.224,-177.565,6.711,148.521
C09928=1191.870,215.538,-60.249,-177.563,6.713,148.521
C09929=1191.865,215.787,-60.273,-177.560,6.715,148.520
C09930=1191.859,216.035,-60.298,-177.557,6.717,148.520
C09931=1191.856,216.284,-60.323,-177.555,6.719,148.520
C09932=1191.851,216.533,-60.348,-177.552,6.721,148.519
C09933=1191.847,216.782,-60.372,-177.550,6.723,148.519
C09934=1191.842,217.031,-60.397,-177.547,6.726,148.519
C09935=1191.837,217.279,-60.422,-177.544,6.728,148.519
C09936=1191.833,217.528,-60.447,-177.541,6.730,148.518
C09937=1191.828,217.776,-60.472,-177.539,6.732,148.518
C09938=1191.824,218.025,-60.497,-177.537,6.734,148.518
C09939=1191.820,218.274,-60.521,-177.533,6.736,148.518
C09940=1191.815,218.523,-60.546,-177.531,6.738,148.517
C09941=1191.810,218.771,-60.572,-177.528,6.740,148.517
C09942=1191.806,219.020,-60.596,-177.526,6.742,148.517
C09943=1191.802,219.268,-60.622,-177.523,6.745,148.517
C09944=1191.796,219.517,-60.646,-177.520,6.747,148.516
C09945=1191.792,219.767,-60.671,-177.518,6.749,148.516
C09946=1191.788,220.014,-60.696,-177.515,6.750,148.516
C09947=1191.783,220.264,-60.721,-177.512,6.753,148.516
C09948=1191.778,220.512,-60.747,-177.510,6.755,148.515
C09949=1191.775,220.761,-60.771,-177.507,6.757,148.515
C09950=1191.770,221.009,-60.796,-177.505,6.759,148.515
C09951=1191.765,221.259,-60.821,-177.502,6.761,148.515
C09952=1191.760,221.507,-60.847,-177.499,6.764,148.514
C09953=1191.756,221.756,-60.872,-177.496,6.765,148.514
C09954=1191.752,222.004,-60.897,-177.494,6.768,148.514
C09955=1191.747,222.253,-60.922,-177.492,6.769,148.513
C09956=1191.742,222.501,-60.947,-177.488,6.772,148.513
C09957=1191.738,222.751,-60.972,-177.486,6.774,148.513
C09958=1191.734,223.000,-60.998,-177.484,6.776,148.513
C09959=1191.729,223.248,-61.022,-177.481,6.778,148.512
C09960=1191.725,223.497,-61.048,-177.478,6.781,148.512
C09961=1191.720,223.745,-61.073,-177.476,6.783,148.512
C09962=1191.716,223.994,-61.098,-177.473,6.784,148.512
C09963=1191.711,224.242,-61.123,-177.471,6.787,148.512
C09964=1191.706,224.492,-61.148,-177.468,6.789,148.511
C09965=1191.702,224.740,-61.174,-177.465,6.791,148.511
C09966=1191.697,224.989,-61.200,-177.463,6.793,148.511
C09967=1191.693,225.237,-61.224,-177.460,6.796,148.511
C09968=1191.689,225.486,-61.249,-177.457,6.798,148.510
C09969=1191.685,225.735,-61.275,-177.455,6.800,148.510
C09970=1191.680,225.983,-61.301,-177.452,6.802,148.510
C09971=1191.675,226.232,-61.326,-177.449,6.805,148.510
C09972=1191.670,226.480,-61.351,-177.447,6.806,148.509
C09973=1191.666,226.729,-61.377,-177.444,6.808,148.509
C09974=1191.662,226.979,-61.402,-177.442,6.810,148.509
C09975=1191.657,227.227,-61.427,-177.439,6.813,148.509
C09976=1191.653,227.476,-61.453,-177.436,6.815,148.508
C09977=1191.648,227.724,-61.478,-177.434,6.817,148.508
C09978=1191.643,227.972,-61.504,-177.431,6.820,148.508
C09979=1191.639,228.222,-61.529,-177.428,6.822,148.508
C09980=1191.634,228.470,-61.554,-177.426,6.824,148.507
C09981=1191.630,228.719,-61.580,-177.423,6.826,148.507
C09982=1191.626,228.968,-61.606,-177.420,6.829,148.507
C09983=1191.621,229.216,-61.631,-177.418,6.830,148.507
C09984=1191.617,229.465,-61.657,-177.416,6.832,148.507
C09985=1191.612,229.713,-61.683,-177.412,6.835,148.506
C09986=1191.607,229.962,-61.707,-177.410,6.837,148.506
C09987=1191.603,230.211,-61.733,-177.408,6.839,148.506
C09988=1191.599,230.460,-61.759,-177.405,6.841,148.506
C09989=1191.594,230.708,-61.784,-177.402,6.844,148.506
C09990=1191.590,230.957,-61.810,-177.400,6.846,148.505
C09991=1191.586,231.205,-61.836,-177.397,6.848,148.505
C09992=1191.581,231.453,-61.861,-177.394,6.851,148.505
C09993=1191.576,231.702,-61.887,-177.392,6.852,148.504
C09994=1191.572,231.951,-61.913,-177.389,6.855,148.504
C09995=1191.567,232.199,-61.939,-177.386,6.857,148.504
C09996=1191.562,232.448,-61.965,-177.384,6.859,148.504
//INST
///DATE 2021/06/25 14:28
///ATTR SC,RW,RJ
////FRAME ROBOT
///GROUP1 RB1
NOP
MOVL C00000 V=800.0 PL=0
MOVL C00001 V=800.0 PL=0
MOVL C00002 V=800.0 PL=0
MOVL C00003 V=800.0 PL=0
MOVL C00004 V=800.0 PL=0
MOVL C00005 V=800.0 PL=0
MOVL C00006 V=800.0 PL=0
MOVL C00007 V=800.0 PL=0
MOVL C00008 V=800.0 PL=0
MOVL C00009 V=800.0 PL=0
MOVL C00010 V=800.0 PL=0
MOVL C00011 V=800.0 PL=0
MOVL C00012 V=800.0 PL=0
MOVL C00013 V=800.0 PL=0
MOVL C00014 V=800.0 PL=0
MOVL C00015 V=800.0 PL=0
MOVL C00016 V=800.0 PL=0
MOVL C00017 V=800.0 PL=0
MOVL C00018 V=800.0 PL=0
MOVL C00019 V=800.0 PL=0
MOVL C00020 V=800.0 PL=0
MOVL C00021 V=800.0 PL=0
MOVL C00022 V=800.0 PL=0
MOVL C00023 V=800.0 PL=0
MOVL C00024 V=800.0 PL=0
MOVL C00025 V=800.0 PL=0
MOVL C00026 V=800.0 PL=0
MOVL C00027 V=800.0 PL=0
MOVL C00028 V=800.0 PL=0
MOVL C00029 V=800.0 PL=0
MOVL C00030 V=800.0 PL=0
MOVL C00031 V=800.0 PL=0
MOVL C00032 V=800.0 PL=0
MOVL C00033 V=800.0 PL=0
MOVL C00034 V=800.0 PL=0
MOVL C00035 V=800.0 PL=0
MOVL C00036 V=800.0 PL=0
MOVL C00037 V=800.0 PL=0
MOVL C00038 V=800.0 PL=0
MOVL C00039 V=800.0 PL=0
MOVL C00040 V=800.0 PL=0
MOVL C00041 V=800.0 PL=0
MOVL C00042 V=800.0 PL=0
MOVL C00043 V=800.0 PL=0
MOVL C00044 V=800.0 PL=0
MOVL C00045 V=800.0 PL=0
MOVL C00046 V=800.0 PL=0
MOVL C00047 V=800.0 PL=0
MOVL C00048 V=800.0 PL=0
MOVL C00049 V=800.0 PL=0
MOVL C00050 V=800.0 PL=0
MOVL C00051 V=800.0 PL=0
MOVL C00052 V=800.0 PL=0
MOVL C00053 V=800.0 PL=0
MOVL C00054 V=800.0 PL=0
MOVL C00055 V=800.0 PL=0
MOVL C00056 V=800.0 PL=0
MOVL C00057 V=800.0 PL=0
MOVL C00058 V=800.0 PL=0
MOVL C00059 V=800.0 PL=0
MOVL C00060 V=800.0 PL=0
MOVL C00061 V=800.0 PL=0
MOVL C00062 V=800.0 PL=0
MOVL C00063 V=800.0 PL=0
MOVL C00064 V=800.0 PL=0
MOVL C00065 V=800.0 PL=0
MOVL C00066 V=800.0 PL=0
MOVL C00067 V=800.0 PL=0
MOVL C00068 V=800.0 PL=0
MOVL C00069 V=800.0 PL=0
MOVL C00070 V=800.0 PL=0
MOVL C00071 V=800.0 PL=0
MOVL C00072 V=800.0 PL=0
MOVL C00073 V=800.0 PL=0
MOVL C00074 V=800.0 PL=0
MOVL C00075 V=800.0 PL=0
MOVL C00076 V=800.0 PL=0
MOVL C00077 V=800.0 PL=0
MOVL C00078 V=800.0 PL=0
MOVL C00079 V=800.0 PL=0
MOVL C00080 V=800.0 PL=0
MOVL C00081 V=800.0 PL=0
MOVL C00082 V=800.0 PL=0
MOVL C00083 V=800.0 PL=0
MOVL C00084 V=800.0 PL=0
MOVL C00085 V=800.0 PL=0
MOVL C00086 V=800.0 PL=0
MOVL C00087 V=800.0 PL=0
MOVL C00088 V=800.0 PL=0
MOVL C00089 V=800.0 PL=0
MOVL C00090 V=800.0 PL=0
MOVL C00091 V=800.0 PL=0
MOVL C00092 V=800.0 PL=0
MOVL C00093 V=800.0 PL=0
MOVL C00094 V=800.0 PL=0
MOVL C00095 V=800.0 PL=0
MOVL C00096 V=800.0 PL=0
MOVL C00097 V=800.0 PL=0
MOVL C00098 V=800.0 PL=0
MOVL C00099 V=800.0 PL=0
MOVL C00100 V=800.0 PL=0
MOVL C00101 V=800.0 PL=0
MOVL C00102 V=800.0 PL=0
MOVL C00103 V=800.0 PL=0
MOVL C00104 V=800.0 PL=0
MOVL C00105 V=800.0 PL=0
MOVL C00106 V=800.0 PL=0
MOVL C00107 V=800.0 PL=0
MOVL C00108 V=800.0 PL=0
MOVL C00109 V=800.0 PL=0
MOVL C00110 V=800.0 PL=0
MOVL C00111 V=800.0 PL=0
MOVL C00112 V=800.0 PL=0
MOVL C00113 V=800.0 PL=0
MOVL C00114 V=800.0 PL=0
MOVL C00115 V=800.0 PL=0
MOVL C00116 V=800.0 PL=0
MOVL C00117 V=800.0 PL=0
MOVL C00118 V=800.0 PL=0
MOVL C00119 V=800.0 PL=0
MOVL C00120 V=800.0 PL=0
MOVL C00121 V=800.0 PL=0
MOVL C00122 V=800.0 PL=0
MOVL C00123 V=800.0 PL=0
MOVL C00124 V=800.0 PL=0
MOVL C00125 V=800.0 PL=0
MOVL C00126 V=800.0 PL=0
MOVL C00127 V=800.0 PL=0
MOVL C00128 V=800.0 PL=0
MOVL C00129 V=800.0 PL=0
MOVL C00130 V=800.0 PL=0
MOVL C00131 V=800.0 PL=0
MOVL C00132 V=800.0 PL=0
MOVL C00133 V=800.0 PL=0
MOVL C00134 V=800.0 PL=0
MOVL C00135 V=800.0 PL=0
MOVL C00136 V=800.0 PL=0
MOVL C00137 V=800.0 PL=0
MOVL C00138 V=800.0 PL=0
MOVL C00139 V=800.0 PL=0
MOVL C00140 V=800.0 PL=0
MOVL C00141 V=800.0 PL=0
MOVL C00142 V=800.0 PL=0
MOVL C00143 V=800.0 PL=0
MOVL C00144 V=800.0 PL=0
MOVL C00145 V=800.0 PL=0
MOVL C00146 V=800.0 PL=0
MOVL C00147 V=800.0 PL=0
MOVL C00148 V=800.0 PL=0
MOVL C00149 V=800.0 PL=0
MOVL C00150 V=800.0 PL=0
MOVL C00151 V=800.0 PL=0
MOVL C00152 V=800.0 PL=0
MOVL C00153 V=800.0 PL=0
MOVL C00154 V=800.0 PL=0
MOVL C00155 V=800.0 PL=0
MOVL C00156 V=800.0 PL=0
MOVL C00157 V=800.0 PL=0
MOVL C00158 V=800.0 PL=0
MOVL C00159 V=800.0 PL=0
MOVL C00160 V=800.0 PL=0
MOVL C00161 V=800.0 PL=0
MOVL C00162 V=800.0 PL=0
MOVL C00163 V=800.0 PL=0
MOVL C00164 V=800.0 PL=0
MOVL C00165 V=800.0 PL=0
MOVL C00166 V=800.0 PL=0
MOVL C00167 V=800.0 PL=0
MOVL C00168 V=800.0 PL=0
MOVL C00169 V=800.0 PL=0
MOVL C00170 V=800.0 PL=0
MOVL C00171 V=800.0 PL=0
MOVL C00172 V=800.0 PL=0
MOVL C00173 V=800.0 PL=0
MOVL C00174 V=800.0 PL=0
MOVL C00175 V=800.0 PL=0
MOVL C00176 V=800.0 PL=0
MOVL C00177 V=800.0 PL=0
MOVL C00178 V=800.0 PL=0
MOVL C00179 V=800.0 PL=0
MOVL C00180 V=800.0 PL=0
MOVL C00181 V=800.0 PL=0
MOVL C00182 V=800.0 PL=0
MOVL C00183 V=800.0 PL=0
MOVL C00184 V=800.0 PL=0
MOVL C00185 V=800.0 PL=0
MOVL C00186 V=800.0 PL=0
MOVL C00187 V=800.0 PL=0
MOVL C00188 V=800.0 PL=0
MOVL C00189 V=800.0 PL=0
MOVL C00190 V=800.0 PL=0
MOVL C00191 V=800.0 PL=0
MOVL C00192 V=800.0 PL=0
MOVL C00193 V=800.0 PL=0
MOVL C00194 V=800.0 PL=0
MOVL C00195 V=800.0 PL=0
MOVL C00196 V=800.0 PL=0
MOVL C00197 V=800.0 PL=0
MOVL C00198 V=800.0 PL=0
MOVL C00199 V=800.0 PL=0
MOVL C00200 V=800.0 PL=0
MOVL C00201 V=800.0 PL=0
MOVL C00202 V=800.0 PL=0
MOVL C00203 V=800.0 PL=0
MOVL C00204 V=800.0 PL=0
MOVL C00205 V=800.0 PL=0
MOVL C00206 V=800.0 PL=0
MOVL C00207 V=800.0 PL=0
MOVL C00208 V=800.0 PL=0
MOVL C00209 V=800.0 PL=0
MOVL C00210 V=800.0 PL=0
MOVL C00211 V=800.0 PL=0
MOVL C00212 V=800.0 PL=0
MOVL C00213 V=800.0 PL=0
MOVL C00214 V=800.0 PL=0
MOVL C00215 V=800.0 PL=0
MOVL C00216 V=800.0 PL=0
MOVL C00217 V=800.0 PL=0
MOVL C00218 V=800.0 PL=0
MOVL C00219 V=800.0 PL=0
MOVL C00220 V=800.0 PL=0
MOVL C00221 V=800.0 PL=0
MOVL C00222 V=800.0 PL=0
MOVL C00223 V=800.0 PL=0
MOVL C00224 V=800.0 PL=0
MOVL C00225 V=800.0 PL=0
MOVL C00226 V=800.0 PL=0
MOVL C00227 V=800.0 PL=0
MOVL C00228 V=800.0 PL=0
MOVL C00229 V=800.0 PL=0
MOVL C00230 V=800.0 PL=0
MOVL C00231 V=800.0 PL=0
MOVL C00232 V=800.0 PL=0
MOVL C00233 V=800.0 PL=0
MOVL C00234 V=800.0 PL=0
MOVL C00235 V=800.0 PL=0
MOVL C00236 V=800.0 PL=0
MOVL C00237 V=800.0 PL=0
MOVL C00238 V=800.0 PL=0
MOVL C00239 V=800.0 PL=0
MOVL C00240 V=800.0 PL=0
MOVL C00241 V=800.0 PL=0
MOVL C00242 V=800.0 PL=0
MOVL C00243 V=800.0 PL=0
MOVL C00244 V=800.0 PL=0
MOVL C00245 V=800.0 PL=0
MOVL C00246 V=800.0 PL=0
MOVL C00247 V=800.0 PL=0
MOVL C00248 V=800.0 PL=0
MOVL C00249 V=800.0 PL=0
MOVL C00250 V=800.0 PL=0
MOVL C00251 V=800.0 PL=0
MOVL C00252 V=800.0 PL=0
MOVL C00253 V=800.0 PL=0
MOVL C00254 V=800.0 PL=0
MOVL C00255 V=800.0 PL=0
MOVL C00256 V=800.0 PL=0
MOVL C00257 V=800.0 PL=0
MOVL C00258 V=800.0 PL=0
MOVL C00259 V=800.0 PL=0
MOVL C00260 V=800.0 PL=0
MOVL C00261 V=800.0 PL=0
MOVL C00262 V=800.0 PL=0
MOVL C00263 V=800.0 PL=0
MOVL C00264 V=800.0 PL=0
MOVL C00265 V=800.0 PL=0
MOVL C00266 V=800.0 PL=0
MOVL C00267 V=800.0 PL=0
MOVL C00268 V=800.0 PL=0
MOVL C00269 V=800.0 PL=0
MOVL C00270 V=800.0 PL=0
MOVL C00271 V=800.0 PL=0
MOVL C00272 V=800.0 PL=0
MOVL C00273 V=800.0 PL=0
MOVL C00274 V=800.0 PL=0
MOVL C00275 V=800.0 PL=0
MOVL C00276 V=800.0 PL=0
MOVL C00277 V=800.0 PL=0
MOVL C00278 V=800.0 PL=0
MOVL C00279 V=800.0 PL=0
MOVL C00280 V=800.0 PL=0
MOVL C00281 V=800.0 PL=0
MOVL C00282 V=800.0 PL=0
MOVL C00283 V=800.0 PL=0
MOVL C00284 V=800.0 PL=0
MOVL C00285 V=800.0 PL=0
MOVL C00286 V=800.0 PL=0
MOVL C00287 V=800.0 PL=0
MOVL C00288 V=800.0 PL=0
MOVL C00289 V=800.0 PL=0
MOVL C00290 V=800.0 PL=0
MOVL C00291 V=800.0 PL=0
MOVL C00292 V=800.0 PL=0
MOVL C00293 V=800.0 PL=0
MOVL C00294 V=800.0 PL=0
MOVL C00295 V=800.0 PL=0
MOVL C00296 V=800.0 PL=0
MOVL C00297 V=800.0 PL=0
MOVL C00298 V=800.0 PL=0
MOVL C00299 V=800.0 PL=0
MOVL C00300 V=800.0 PL=0
MOVL C00301 V=800.0 PL=0
MOVL C00302 V=800.0 PL=0
MOVL C00303 V=800.0 PL=0
MOVL C00304 V=800.0 PL=0
MOVL C00305 V=800.0 PL=0
MOVL C00306 V=800.0 PL=0
MOVL C00307 V=800.0 PL=0
MOVL C00308 V=800.0 PL=0
MOVL C00309 V=800.0 PL=0
MOVL C00310 V=800.0 PL=0
MOVL C00311 V=800.0 PL=0
MOVL C00312 V=800.0 PL=0
MOVL C00313 V=800.0 PL=0
MOVL C00314 V=800.0 PL=0
MOVL C00315 V=800.0 PL=0
MOVL C00316 V=800.0 PL=0
MOVL C00317 V=800.0 PL=0
MOVL C00318 V=800.0 PL=0
MOVL C00319 V=800.0 PL=0
MOVL C00320 V=800.0 PL=0
MOVL C00321 V=800.0 PL=0
MOVL C00322 V=800.0 PL=0
MOVL C00323 V=800.0 PL=0
MOVL C00324 V=800.0 PL=0
MOVL C00325 V=800.0 PL=0
MOVL C00326 V=800.0 PL=0
MOVL C00327 V=800.0 PL=0
MOVL C00328 V=800.0 PL=0
MOVL C00329 V=800.0 PL=0
MOVL C00330 V=800.0 PL=0
MOVL C00331 V=800.0 PL=0
MOVL C00332 V=800.0 PL=0
MOVL C00333 V=800.0 PL=0
MOVL C00334 V=800.0 PL=0
MOVL C00335 V=800.0 PL=0
MOVL C00336 V=800.0 PL=0
MOVL C00337 V=800.0 PL=0
MOVL C00338 V=800.0 PL=0
MOVL C00339 V=800.0 PL=0
MOVL C00340 V=800.0 PL=0
MOVL C00341 V=800.0 PL=0
MOVL C00342 V=800.0 PL=0
MOVL C00343 V=800.0 PL=0
MOVL C00344 V=800.0 PL=0
MOVL C00345 V=800.0 PL=0
MOVL C00346 V=800.0 PL=0
MOVL C00347 V=800.0 PL=0
MOVL C00348 V=800.0 PL=0
MOVL C00349 V=800.0 PL=0
MOVL C00350 V=800.0 PL=0
MOVL C00351 V=800.0 PL=0
MOVL C00352 V=800.0 PL=0
MOVL C00353 V=800.0 PL=0
MOVL C00354 V=800.0 PL=0
MOVL C00355 V=800.0 PL=0
MOVL C00356 V=800.0 PL=0
MOVL C00357 V=800.0 PL=0
MOVL C00358 V=800.0 PL=0
MOVL C00359 V=800.0 PL=0
MOVL C00360 V=800.0 PL=0
MOVL C00361 V=800.0 PL=0
MOVL C00362 V=800.0 PL=0
MOVL C00363 V=800.0 PL=0
MOVL C00364 V=800.0 PL=0
MOVL C00365 V=800.0 PL=0
MOVL C00366 V=800.0 PL=0
MOVL C00367 V=800.0 PL=0
MOVL C00368 V=800.0 PL=0
MOVL C00369 V=800.0 PL=0
MOVL C00370 V=800.0 PL=0
MOVL C00371 V=800.0 PL=0
MOVL C00372 V=800.0 PL=0
MOVL C00373 V=800.0 PL=0
MOVL C00374 V=800.0 PL=0
MOVL C00375 V=800.0 PL=0
MOVL C00376 V=800.0 PL=0
MOVL C00377 V=800.0 PL=0
MOVL C00378 V=800.0 PL=0
MOVL C00379 V=800.0 PL=0
MOVL C00380 V=800.0 PL=0
MOVL C00381 V=800.0 PL=0
MOVL C00382 V=800.0 PL=0
MOVL C00383 V=800.0 PL=0
MOVL C00384 V=800.0 PL=0
MOVL C00385 V=800.0 PL=0
MOVL C00386 V=800.0 PL=0
MOVL C00387 V=800.0 PL=0
MOVL C00388 V=800.0 PL=0
MOVL C00389 V=800.0 PL=0
MOVL C00390 V=800.0 PL=0
MOVL C00391 V=800.0 PL=0
MOVL C00392 V=800.0 PL=0
MOVL C00393 V=800.0 PL=0
MOVL C00394 V=800.0 PL=0
MOVL C00395 V=800.0 PL=0
MOVL C00396 V=800.0 PL=0
MOVL C00397 V=800.0 PL=0
MOVL C00398 V=800.0 PL=0
MOVL C00399 V=800.0 PL=0
MOVL C00400 V=800.0 PL=0
MOVL C00401 V=800.0 PL=0
MOVL C00402 V=800.0 PL=0
MOVL C00403 V=800.0 PL=0
MOVL C00404 V=800.0 PL=0
MOVL C00405 V=800.0 PL=0
MOVL C00406 V=800.0 PL=0
MOVL C00407 V=800.0 PL=0
MOVL C00408 V=800.0 PL=0
MOVL C00409 V=800.0 PL=0
MOVL C00410 V=800.0 PL=0
MOVL C00411 V=800.0 PL=0
MOVL C00412 V=800.0 PL=0
MOVL C00413 V=800.0 PL=0
MOVL C00414 V=800.0 PL=0
MOVL C00415 V=800.0 PL=0
MOVL C00416 V=800.0 PL=0
MOVL C00417 V=800.0 PL=0
MOVL C00418 V=800.0 PL=0
MOVL C00419 V=800.0 PL=0
MOVL C00420 V=800.0 PL=0
MOVL C00421 V=800.0 PL=0
MOVL C00422 V=800.0 PL=0
MOVL C00423 V=800.0 PL=0
MOVL C00424 V=800.0 PL=0
MOVL C00425 V=800.0 PL=0
MOVL C00426 V=800.0 PL=0
MOVL C00427 V=800.0 PL=0
MOVL C00428 V=800.0 PL=0
MOVL C00429 V=800.0 PL=0
MOVL C00430 V=800.0 PL=0
MOVL C00431 V=800.0 PL=0
MOVL C00432 V=800.0 PL=0
MOVL C00433 V=800.0 PL=0
MOVL C00434 V=800.0 PL=0
MOVL C00435 V=800.0 PL=0
MOVL C00436 V=800.0 PL=0
MOVL C00437 V=800.0 PL=0
MOVL C00438 V=800.0 PL=0
MOVL C00439 V=800.0 PL=0
MOVL C00440 V=800.0 PL=0
MOVL C00441 V=800.0 PL=0
MOVL C00442 V=800.0 PL=0
MOVL C00443 V=800.0 PL=0
MOVL C00444 V=800.0 PL=0
MOVL C00445 V=800.0 PL=0
MOVL C00446 V=800.0 PL=0
MOVL C00447 V=800.0 PL=0
MOVL C00448 V=800.0 PL=0
MOVL C00449 V=800.0 PL=0
MOVL C00450 V=800.0 PL=0
MOVL C00451 V=800.0 PL=0
MOVL C00452 V=800.0 PL=0
MOVL C00453 V=800.0 PL=0
MOVL C00454 V=800.0 PL=0
MOVL C00455 V=800.0 PL=0
MOVL C00456 V=800.0 PL=0
MOVL C00457 V=800.0 PL=0
MOVL C00458 V=800.0 PL=0
MOVL C00459 V=800.0 PL=0
MOVL C00460 V=800.0 PL=0
MOVL C00461 V=800.0 PL=0
MOVL C00462 V=800.0 PL=0
MOVL C00463 V=800.0 PL=0
MOVL C00464 V=800.0 PL=0
MOVL C00465 V=800.0 PL=0
MOVL C00466 V=800.0 PL=0
MOVL C00467 V=800.0 PL=0
MOVL C00468 V=800.0 PL=0
MOVL C00469 V=800.0 PL=0
MOVL C00470 V=800.0 PL=0
MOVL C00471 V=800.0 PL=0
MOVL C00472 V=800.0 PL=0
MOVL C00473 V=800.0 PL=0
MOVL C00474 V=800.0 PL=0
MOVL C00475 V=800.0 PL=0
MOVL C00476 V=800.0 PL=0
MOVL C00477 V=800.0 PL=0
MOVL C00478 V=800.0 PL=0
MOVL C00479 V=800.0 PL=0
MOVL C00480 V=800.0 PL=0
MOVL C00481 V=800.0 PL=0
MOVL C00482 V=800.0 PL=0
MOVL C00483 V=800.0 PL=0
MOVL C00484 V=800.0 PL=0
MOVL C00485 V=800.0 PL=0
MOVL C00486 V=800.0 PL=0
MOVL C00487 V=800.0 PL=0
MOVL C00488 V=800.0 PL=0
MOVL C00489 V=800.0 PL=0
MOVL C00490 V=800.0 PL=0
MOVL C00491 V=800.0 PL=0
MOVL C00492 V=800.0 PL=0
MOVL C00493 V=800.0 PL=0
MOVL C00494 V=800.0 PL=0
MOVL C00495 V=800.0 PL=0
MOVL C00496 V=800.0 PL=0
MOVL C00497 V=800.0 PL=0
MOVL C00498 V=800.0 PL=0
MOVL C00499 V=800.0 PL=0
MOVL C00500 V=800.0 PL=0
MOVL C00501 V=800.0 PL=0
MOVL C00502 V=800.0 PL=0
MOVL C00503 V=800.0 PL=0
MOVL C00504 V=800.0 PL=0
MOVL C00505 V=800.0 PL=0
MOVL C00506 V=800.0 PL=0
MOVL C00507 V=800.0 PL=0
MOVL C00508 V=800.0 PL=0
MOVL C00509 V=800.0 PL=0
MOVL C00510 V=800.0 PL=0
MOVL C00511 V=800.0 PL=0
MOVL C00512 V=800.0 PL=0
MOVL C00513 V=800.0 PL=0
MOVL C00514 V=800.0 PL=0
MOVL C00515 V=800.0 PL=0
MOVL C00516 V=800.0 PL=0
MOVL C00517 V=800.0 PL=0
MOVL C00518 V=800.0 PL=0
MOVL C00519 V=800.0 PL=0
MOVL C00520 V=800.0 PL=0
MOVL C00521 V=800.0 PL=0
MOVL C00522 V=800.0 PL=0
MOVL C00523 V=800.0 PL=0
MOVL C00524 V=800.0 PL=0
MOVL C00525 V=800.0 PL=0
MOVL C00526 V=800.0 PL=0
MOVL C00527 V=800.0 PL=0
MOVL C00528 V=800.0 PL=0
MOVL C00529 V=800.0 PL=0
MOVL C00530 V=800.0 PL=0
MOVL C00531 V=800.0 PL=0
MOVL C00532 V=800.0 PL=0
MOVL C00533 V=800.0 PL=0
MOVL C00534 V=800.0 PL=0
MOVL C00535 V=800.0 PL=0
MOVL C00536 V=800.0 PL=0
MOVL C00537 V=800.0 PL=0
MOVL C00538 V=800.0 PL=0
MOVL C00539 V=800.0 PL=0
MOVL C00540 V=800.0 PL=0
MOVL C00541 V=800.0 PL=0
MOVL C00542 V=800.0 PL=0
MOVL C00543 V=800.0 PL=0
MOVL C00544 V=800.0 PL=0
MOVL C00545 V=800.0 PL=0
MOVL C00546 V=800.0 PL=0
MOVL C00547 V=800.0 PL=0
MOVL C00548 V=800.0 PL=0
MOVL C00549 V=800.0 PL=0
MOVL C00550 V=800.0 PL=0
MOVL C00551 V=800.0 PL=0
MOVL C00552 V=800.0 PL=0
MOVL C00553 V=800.0 PL=0
MOVL C00554 V=800.0 PL=0
MOVL C00555 V=800.0 PL=0
MOVL C00556 V=800.0 PL=0
MOVL C00557 V=800.0 PL=0
MOVL C00558 V=800.0 PL=0
MOVL C00559 V=800.0 PL=0
MOVL C00560 V=800.0 PL=0
MOVL C00561 V=800.0 PL=0
MOVL C00562 V=800.0 PL=0
MOVL C00563 V=800.0 PL=0
MOVL C00564 V=800.0 PL=0
MOVL C00565 V=800.0 PL=0
MOVL C00566 V=800.0 PL=0
MOVL C00567 V=800.0 PL=0
MOVL C00568 V=800.0 PL=0
MOVL C00569 V=800.0 PL=0
MOVL C00570 V=800.0 PL=0
MOVL C00571 V=800.0 PL=0
MOVL C00572 V=800.0 PL=0
MOVL C00573 V=800.0 PL=0
MOVL C00574 V=800.0 PL=0
MOVL C00575 V=800.0 PL=0
MOVL C00576 V=800.0 PL=0
MOVL C00577 V=800.0 PL=0
MOVL C00578 V=800.0 PL=0
MOVL C00579 V=800.0 PL=0
MOVL C00580 V=800.0 PL=0
MOVL C00581 V=800.0 PL=0
MOVL C00582 V=800.0 PL=0
MOVL C00583 V=800.0 PL=0
MOVL C00584 V=800.0 PL=0
MOVL C00585 V=800.0 PL=0
MOVL C00586 V=800.0 PL=0
MOVL C00587 V=800.0 PL=0
MOVL C00588 V=800.0 PL=0
MOVL C00589 V=800.0 PL=0
MOVL C00590 V=800.0 PL=0
MOVL C00591 V=800.0 PL=0
MOVL C00592 V=800.0 PL=0
MOVL C00593 V=800.0 PL=0
MOVL C00594 V=800.0 PL=0
MOVL C00595 V=800.0 PL=0
MOVL C00596 V=800.0 PL=0
MOVL C00597 V=800.0 PL=0
MOVL C00598 V=800.0 PL=0
MOVL C00599 V=800.0 PL=0
MOVL C00600 V=800.0 PL=0
MOVL C00601 V=800.0 PL=0
MOVL C00602 V=800.0 PL=0
MOVL C00603 V=800.0 PL=0
MOVL C00604 V=800.0 PL=0
MOVL C00605 V=800.0 PL=0
MOVL C00606 V=800.0 PL=0
MOVL C00607 V=800.0 PL=0
MOVL C00608 V=800.0 PL=0
MOVL C00609 V=800.0 PL=0
MOVL C00610 V=800.0 PL=0
MOVL C00611 V=800.0 PL=0
MOVL C00612 V=800.0 PL=0
MOVL C00613 V=800.0 PL=0
MOVL C00614 V=800.0 PL=0
MOVL C00615 V=800.0 PL=0
MOVL C00616 V=800.0 PL=0
MOVL C00617 V=800.0 PL=0
MOVL C00618 V=800.0 PL=0
MOVL C00619 V=800.0 PL=0
MOVL C00620 V=800.0 PL=0
MOVL C00621 V=800.0 PL=0
MOVL C00622 V=800.0 PL=0
MOVL C00623 V=800.0 PL=0
MOVL C00624 V=800.0 PL=0
MOVL C00625 V=800.0 PL=0
MOVL C00626 V=800.0 PL=0
MOVL C00627 V=800.0 PL=0
MOVL C00628 V=800.0 PL=0
MOVL C00629 V=800.0 PL=0
MOVL C00630 V=800.0 PL=0
MOVL C00631 V=800.0 PL=0
MOVL C00632 V=800.0 PL=0
MOVL C00633 V=800.0 PL=0
MOVL C00634 V=800.0 PL=0
MOVL C00635 V=800.0 PL=0
MOVL C00636 V=800.0 PL=0
MOVL C00637 V=800.0 PL=0
MOVL C00638 V=800.0 PL=0
MOVL C00639 V=800.0 PL=0
MOVL C00640 V=800.0 PL=0
MOVL C00641 V=800.0 PL=0
MOVL C00642 V=800.0 PL=0
MOVL C00643 V=800.0 PL=0
MOVL C00644 V=800.0 PL=0
MOVL C00645 V=800.0 PL=0
MOVL C00646 V=800.0 PL=0
MOVL C00647 V=800.0 PL=0
MOVL C00648 V=800.0 PL=0
MOVL C00649 V=800.0 PL=0
MOVL C00650 V=800.0 PL=0
MOVL C00651 V=800.0 PL=0
MOVL C00652 V=800.0 PL=0
MOVL C00653 V=800.0 PL=0
MOVL C00654 V=800.0 PL=0
MOVL C00655 V=800.0 PL=0
MOVL C00656 V=800.0 PL=0
MOVL C00657 V=800.0 PL=0
MOVL C00658 V=800.0 PL=0
MOVL C00659 V=800.0 PL=0
MOVL C00660 V=800.0 PL=0
MOVL C00661 V=800.0 PL=0
MOVL C00662 V=800.0 PL=0
MOVL C00663 V=800.0 PL=0
MOVL C00664 V=800.0 PL=0
MOVL C00665 V=800.0 PL=0
MOVL C00666 V=800.0 PL=0
MOVL C00667 V=800.0 PL=0
MOVL C00668 V=800.0 PL=0
MOVL C00669 V=800.0 PL=0
MOVL C00670 V=800.0 PL=0
MOVL C00671 V=800.0 PL=0
MOVL C00672 V=800.0 PL=0
MOVL C00673 V=800.0 PL=0
MOVL C00674 V=800.0 PL=0
MOVL C00675 V=800.0 PL=0
MOVL C00676 V=800.0 PL=0
MOVL C00677 V=800.0 PL=0
MOVL C00678 V=800.0 PL=0
MOVL C00679 V=800.0 PL=0
MOVL C00680 V=800.0 PL=0
MOVL C00681 V=800.0 PL=0
MOVL C00682 V=800.0 PL=0
MOVL C00683 V=800.0 PL=0
MOVL C00684 V=800.0 PL=0
MOVL C00685 V=800.0 PL=0
MOVL C00686 V=800.0 PL=0
MOVL C00687 V=800.0 PL=0
MOVL C00688 V=800.0 PL=0
MOVL C00689 V=800.0 PL=0
MOVL C00690 V=800.0 PL=0
MOVL C00691 V=800.0 PL=0
MOVL C00692 V=800.0 PL=0
MOVL C00693 V=800.0 PL=0
MOVL C00694 V=800.0 PL=0
MOVL C00695 V=800.0 PL=0
MOVL C00696 V=800.0 PL=0
MOVL C00697 V=800.0 PL=0
MOVL C00698 V=800.0 PL=0
MOVL C00699 V=800.0 PL=0
MOVL C00700 V=800.0 PL=0
MOVL C00701 V=800.0 PL=0
MOVL C00702 V=800.0 PL=0
MOVL C00703 V=800.0 PL=0
MOVL C00704 V=800.0 PL=0
MOVL C00705 V=800.0 PL=0
MOVL C00706 V=800.0 PL=0
MOVL C00707 V=800.0 PL=0
MOVL C00708 V=800.0 PL=0
MOVL C00709 V=800.0 PL=0
MOVL C00710 V=800.0 PL=0
MOVL C00711 V=800.0 PL=0
MOVL C00712 V=800.0 PL=0
MOVL C00713 V=800.0 PL=0
MOVL C00714 V=800.0 PL=0
MOVL C00715 V=800.0 PL=0
MOVL C00716 V=800.0 PL=0
MOVL C00717 V=800.0 PL=0
MOVL C00718 V=800.0 PL=0
MOVL C00719 V=800.0 PL=0
MOVL C00720 V=800.0 PL=0
MOVL C00721 V=800.0 PL=0
MOVL C00722 V=800.0 PL=0
MOVL C00723 V=800.0 PL=0
MOVL C00724 V=800.0 PL=0
MOVL C00725 V=800.0 PL=0
MOVL C00726 V=800.0 PL=0
MOVL C00727 V=800.0 PL=0
MOVL C00728 V=800.0 PL=0
MOVL C00729 V=800.0 PL=0
MOVL C00730 V=800.0 PL=0
MOVL C00731 V=800.0 PL=0
MOVL C00732 V=800.0 PL=0
MOVL C00733 V=800.0 PL=0
MOVL C00734 V=800.0 PL=0
MOVL C00735 V=800.0 PL=0
MOVL C00736 V=800.0 PL=0
MOVL C00737 V=800.0 PL=0
MOVL C00738 V=800.0 PL=0
MOVL C00739 V=800.0 PL=0
MOVL C00740 V=800.0 PL=0
MOVL C00741 V=800.0 PL=0
MOVL C00742 V=800.0 PL=0
MOVL C00743 V=800.0 PL=0
MOVL C00744 V=800.0 PL=0
MOVL C00745 V=800.0 PL=0
MOVL C00746 V=800.0 PL=0
MOVL C00747 V=800.0 PL=0
MOVL C00748 V=800.0 PL=0
MOVL C00749 V=800.0 PL=0
MOVL C00750 V=800.0 PL=0
MOVL C00751 V=800.0 PL=0
MOVL C00752 V=800.0 PL=0
MOVL C00753 V=800.0 PL=0
MOVL C00754 V=800.0 PL=0
MOVL C00755 V=800.0 PL=0
MOVL C00756 V=800.0 PL=0
MOVL C00757 V=800.0 PL=0
MOVL C00758 V=800.0 PL=0
MOVL C00759 V=800.0 PL=0
MOVL C00760 V=800.0 PL=0
MOVL C00761 V=800.0 PL=0
MOVL C00762 V=800.0 PL=0
MOVL C00763 V=800.0 PL=0
MOVL C00764 V=800.0 PL=0
MOVL C00765 V=800.0 PL=0
MOVL C00766 V=800.0 PL=0
MOVL C00767 V=800.0 PL=0
MOVL C00768 V=800.0 PL=0
MOVL C00769 V=800.0 PL=0
MOVL C00770 V=800.0 PL=0
MOVL C00771 V=800.0 PL=0
MOVL C00772 V=800.0 PL=0
MOVL C00773 V=800.0 PL=0
MOVL C00774 V=800.0 PL=0
MOVL C00775 V=800.0 PL=0
MOVL C00776 V=800.0 PL=0
MOVL C00777 V=800.0 PL=0
MOVL C00778 V=800.0 PL=0
MOVL C00779 V=800.0 PL=0
MOVL C00780 V=800.0 PL=0
MOVL C00781 V=800.0 PL=0
MOVL C00782 V=800.0 PL=0
MOVL C00783 V=800.0 PL=0
MOVL C00784 V=800.0 PL=0
MOVL C00785 V=800.0 PL=0
MOVL C00786 V=800.0 PL=0
MOVL C00787 V=800.0 PL=0
MOVL C00788 V=800.0 PL=0
MOVL C00789 V=800.0 PL=0
MOVL C00790 V=800.0 PL=0
MOVL C00791 V=800.0 PL=0
MOVL C00792 V=800.0 PL=0
MOVL C00793 V=800.0 PL=0
MOVL C00794 V=800.0 PL=0
MOVL C00795 V=800.0 PL=0
MOVL C00796 V=800.0 PL=0
MOVL C00797 V=800.0 PL=0
MOVL C00798 V=800.0 PL=0
MOVL C00799 V=800.0 PL=0
MOVL C00800 V=800.0 PL=0
MOVL C00801 V=800.0 PL=0
MOVL C00802 V=800.0 PL=0
MOVL C00803 V=800.0 PL=0
MOVL C00804 V=800.0 PL=0
MOVL C00805 V=800.0 PL=0
MOVL C00806 V=800.0 PL=0
MOVL C00807 V=800.0 PL=0
MOVL C00808 V=800.0 PL=0
MOVL C00809 V=800.0 PL=0
MOVL C00810 V=800.0 PL=0
MOVL C00811 V=800.0 PL=0
MOVL C00812 V=800.0 PL=0
MOVL C00813 V=800.0 PL=0
MOVL C00814 V=800.0 PL=0
MOVL C00815 V=800.0 PL=0
MOVL C00816 V=800.0 PL=0
MOVL C00817 V=800.0 PL=0
MOVL C00818 V=800.0 PL=0
MOVL C00819 V=800.0 PL=0
MOVL C00820 V=800.0 PL=0
MOVL C00821 V=800.0 PL=0
MOVL C00822 V=800.0 PL=0
MOVL C00823 V=800.0 PL=0
MOVL C00824 V=800.0 PL=0
MOVL C00825 V=800.0 PL=0
MOVL C00826 V=800.0 PL=0
MOVL C00827 V=800.0 PL=0
MOVL C00828 V=800.0 PL=0
MOVL C00829 V=800.0 PL=0
MOVL C00830 V=800.0 PL=0
MOVL C00831 V=800.0 PL=0
MOVL C00832 V=800.0 PL=0
MOVL C00833 V=800.0 PL=0
MOVL C00834 V=800.0 PL=0
MOVL C00835 V=800.0 PL=0
MOVL C00836 V=800.0 PL=0
MOVL C00837 V=800.0 PL=0
MOVL C00838 V=800.0 PL=0
MOVL C00839 V=800.0 PL=0
MOVL C00840 V=800.0 PL=0
MOVL C00841 V=800.0 PL=0
MOVL C00842 V=800.0 PL=0
MOVL C00843 V=800.0 PL=0
MOVL C00844 V=800.0 PL=0
MOVL C00845 V=800.0 PL=0
MOVL C00846 V=800.0 PL=0
MOVL C00847 V=800.0 PL=0
MOVL C00848 V=800.0 PL=0
MOVL C00849 V=800.0 PL=0
MOVL C00850 V=800.0 PL=0
MOVL C00851 V=800.0 PL=0
MOVL C00852 V=800.0 PL=0
MOVL C00853 V=800.0 PL=0
MOVL C00854 V=800.0 PL=0
MOVL C00855 V=800.0 PL=0
MOVL C00856 V=800.0 PL=0
MOVL C00857 V=800.0 PL=0
MOVL C00858 V=800.0 PL=0
MOVL C00859 V=800.0 PL=0
MOVL C00860 V=800.0 PL=0
MOVL C00861 V=800.0 PL=0
MOVL C00862 V=800.0 PL=0
MOVL C00863 V=800.0 PL=0
MOVL C00864 V=800.0 PL=0
MOVL C00865 V=800.0 PL=0
MOVL C00866 V=800.0 PL=0
MOVL C00867 V=800.0 PL=0
MOVL C00868 V=800.0 PL=0
MOVL C00869 V=800.0 PL=0
MOVL C00870 V=800.0 PL=0
MOVL C00871 V=800.0 PL=0
MOVL C00872 V=800.0 PL=0
MOVL C00873 V=800.0 PL=0
MOVL C00874 V=800.0 PL=0
MOVL C00875 V=800.0 PL=0
MOVL C00876 V=800.0 PL=0
MOVL C00877 V=800.0 PL=0
MOVL C00878 V=800.0 PL=0
MOVL C00879 V=800.0 PL=0
MOVL C00880 V=800.0 PL=0
MOVL C00881 V=800.0 PL=0
MOVL C00882 V=800.0 PL=0
MOVL C00883 V=800.0 PL=0
MOVL C00884 V=800.0 PL=0
MOVL C00885 V=800.0 PL=0
MOVL C00886 V=800.0 PL=0
MOVL C00887 V=800.0 PL=0
MOVL C00888 V=800.0 PL=0
MOVL C00889 V=800.0 PL=0
MOVL C00890 V=800.0 PL=0
MOVL C00891 V=800.0 PL=0
MOVL C00892 V=800.0 PL=0
MOVL C00893 V=800.0 PL=0
MOVL C00894 V=800.0 PL=0
MOVL C00895 V=800.0 PL=0
MOVL C00896 V=800.0 PL=0
MOVL C00897 V=800.0 PL=0
MOVL C00898 V=800.0 PL=0
MOVL C00899 V=800.0 PL=0
MOVL C00900 V=800.0 PL=0
MOVL C00901 V=800.0 PL=0
MOVL C00902 V=800.0 PL=0
MOVL C00903 V=800.0 PL=0
MOVL C00904 V=800.0 PL=0
MOVL C00905 V=800.0 PL=0
MOVL C00906 V=800.0 PL=0
MOVL C00907 V=800.0 PL=0
MOVL C00908 V=800.0 PL=0
MOVL C00909 V=800.0 PL=0
MOVL C00910 V=800.0 PL=0
MOVL C00911 V=800.0 PL=0
MOVL C00912 V=800.0 PL=0
MOVL C00913 V=800.0 PL=0
MOVL C00914 V=800.0 PL=0
MOVL C00915 V=800.0 PL=0
MOVL C00916 V=800.0 PL=0
MOVL C00917 V=800.0 PL=0
MOVL C00918 V=800.0 PL=0
MOVL C00919 V=800.0 PL=0
MOVL C00920 V=800.0 PL=0
MOVL C00921 V=800.0 PL=0
MOVL C00922 V=800.0 PL=0
MOVL C00923 V=800.0 PL=0
MOVL C00924 V=800.0 PL=0
MOVL C00925 V=800.0 PL=0
MOVL C00926 V=800.0 PL=0
MOVL C00927 V=800.0 PL=0
MOVL C00928 V=800.0 PL=0
MOVL C00929 V=800.0 PL=0
MOVL C00930 V=800.0 PL=0
MOVL C00931 V=800.0 PL=0
MOVL C00932 V=800.0 PL=0
MOVL C00933 V=800.0 PL=0
MOVL C00934 V=800.0 PL=0
MOVL C00935 V=800.0 PL=0
MOVL C00936 V=800.0 PL=0
MOVL C00937 V=800.0 PL=0
MOVL C00938 V=800.0 PL=0
MOVL C00939 V=800.0 PL=0
MOVL C00940 V=800.0 PL=0
MOVL C00941 V=800.0 PL=0
MOVL C00942 V=800.0 PL=0
MOVL C00943 V=800.0 PL=0
MOVL C00944 V=800.0 PL=0
MOVL C00945 V=800.0 PL=0
MOVL C00946 V=800.0 PL=0
MOVL C00947 V=800.0 PL=0
MOVL C00948 V=800.0 PL=0
MOVL C00949 V=800.0 PL=0
MOVL C00950 V=800.0 PL=0
MOVL C00951 V=800.0 PL=0
MOVL C00952 V=800.0 PL=0
MOVL C00953 V=800.0 PL=0
MOVL C00954 V=800.0 PL=0
MOVL C00955 V=800.0 PL=0
MOVL C00956 V=800.0 PL=0
MOVL C00957 V=800.0 PL=0
MOVL C00958 V=800.0 PL=0
MOVL C00959 V=800.0 PL=0
MOVL C00960 V=800.0 PL=0
MOVL C00961 V=800.0 PL=0
MOVL C00962 V=800.0 PL=0
MOVL C00963 V=800.0 PL=0
MOVL C00964 V=800.0 PL=0
MOVL C00965 V=800.0 PL=0
MOVL C00966 V=800.0 PL=0
MOVL C00967 V=800.0 PL=0
MOVL C00968 V=800.0 PL=0
MOVL C00969 V=800.0 PL=0
MOVL C00970 V=800.0 PL=0
MOVL C00971 V=800.0 PL=0
MOVL C00972 V=800.0 PL=0
MOVL C00973 V=800.0 PL=0
MOVL C00974 V=800.0 PL=0
MOVL C00975 V=800.0 PL=0
MOVL C00976 V=800.0 PL=0
MOVL C00977 V=800.0 PL=0
MOVL C00978 V=800.0 PL=0
MOVL C00979 V=800.0 PL=0
MOVL C00980 V=800.0 PL=0
MOVL C00981 V=800.0 PL=0
MOVL C00982 V=800.0 PL=0
MOVL C00983 V=800.0 PL=0
MOVL C00984 V=800.0 PL=0
MOVL C00985 V=800.0 PL=0
MOVL C00986 V=800.0 PL=0
MOVL C00987 V=800.0 PL=0
MOVL C00988 V=800.0 PL=0
MOVL C00989 V=800.0 PL=0
MOVL C00990 V=800.0 PL=0
MOVL C00991 V=800.0 PL=0
MOVL C00992 V=800.0 PL=0
MOVL C00993 V=800.0 PL=0
MOVL C00994 V=800.0 PL=0
MOVL C00995 V=800.0 PL=0
MOVL C00996 V=800.0 PL=0
MOVL C00997 V=800.0 PL=0
MOVL C00998 V=800.0 PL=0
MOVL C00999 V=800.0 PL=0
MOVL C01000 V=800.0 PL=0
MOVL C01001 V=800.0 PL=0
MOVL C01002 V=800.0 PL=0
MOVL C01003 V=800.0 PL=0
MOVL C01004 V=800.0 PL=0
MOVL C01005 V=800.0 PL=0
MOVL C01006 V=800.0 PL=0
MOVL C01007 V=800.0 PL=0
MOVL C01008 V=800.0 PL=0
MOVL C01009 V=800.0 PL=0
MOVL C01010 V=800.0 PL=0
MOVL C01011 V=800.0 PL=0
MOVL C01012 V=800.0 PL=0
MOVL C01013 V=800.0 PL=0
MOVL C01014 V=800.0 PL=0
MOVL C01015 V=800.0 PL=0
MOVL C01016 V=800.0 PL=0
MOVL C01017 V=800.0 PL=0
MOVL C01018 V=800.0 PL=0
MOVL C01019 V=800.0 PL=0
MOVL C01020 V=800.0 PL=0
MOVL C01021 V=800.0 PL=0
MOVL C01022 V=800.0 PL=0
MOVL C01023 V=800.0 PL=0
MOVL C01024 V=800.0 PL=0
MOVL C01025 V=800.0 PL=0
MOVL C01026 V=800.0 PL=0
MOVL C01027 V=800.0 PL=0
MOVL C01028 V=800.0 PL=0
MOVL C01029 V=800.0 PL=0
MOVL C01030 V=800.0 PL=0
MOVL C01031 V=800.0 PL=0
MOVL C01032 V=800.0 PL=0
MOVL C01033 V=800.0 PL=0
MOVL C01034 V=800.0 PL=0
MOVL C01035 V=800.0 PL=0
MOVL C01036 V=800.0 PL=0
MOVL C01037 V=800.0 PL=0
MOVL C01038 V=800.0 PL=0
MOVL C01039 V=800.0 PL=0
MOVL C01040 V=800.0 PL=0
MOVL C01041 V=800.0 PL=0
MOVL C01042 V=800.0 PL=0
MOVL C01043 V=800.0 PL=0
MOVL C01044 V=800.0 PL=0
MOVL C01045 V=800.0 PL=0
MOVL C01046 V=800.0 PL=0
MOVL C01047 V=800.0 PL=0
MOVL C01048 V=800.0 PL=0
MOVL C01049 V=800.0 PL=0
MOVL C01050 V=800.0 PL=0
MOVL C01051 V=800.0 PL=0
MOVL C01052 V=800.0 PL=0
MOVL C01053 V=800.0 PL=0
MOVL C01054 V=800.0 PL=0
MOVL C01055 V=800.0 PL=0
MOVL C01056 V=800.0 PL=0
MOVL C01057 V=800.0 PL=0
MOVL C01058 V=800.0 PL=0
MOVL C01059 V=800.0 PL=0
MOVL C01060 V=800.0 PL=0
MOVL C01061 V=800.0 PL=0
MOVL C01062 V=800.0 PL=0
MOVL C01063 V=800.0 PL=0
MOVL C01064 V=800.0 PL=0
MOVL C01065 V=800.0 PL=0
MOVL C01066 V=800.0 PL=0
MOVL C01067 V=800.0 PL=0
MOVL C01068 V=800.0 PL=0
MOVL C01069 V=800.0 PL=0
MOVL C01070 V=800.0 PL=0
MOVL C01071 V=800.0 PL=0
MOVL C01072 V=800.0 PL=0
MOVL C01073 V=800.0 PL=0
MOVL C01074 V=800.0 PL=0
MOVL C01075 V=800.0 PL=0
MOVL C01076 V=800.0 PL=0
MOVL C01077 V=800.0 PL=0
MOVL C01078 V=800.0 PL=0
MOVL C01079 V=800.0 PL=0
MOVL C01080 V=800.0 PL=0
MOVL C01081 V=800.0 PL=0
MOVL C01082 V=800.0 PL=0
MOVL C01083 V=800.0 PL=0
MOVL C01084 V=800.0 PL=0
MOVL C01085 V=800.0 PL=0
MOVL C01086 V=800.0 PL=0
MOVL C01087 V=800.0 PL=0
MOVL C01088 V=800.0 PL=0
MOVL C01089 V=800.0 PL=0
MOVL C01090 V=800.0 PL=0
MOVL C01091 V=800.0 PL=0
MOVL C01092 V=800.0 PL=0
MOVL C01093 V=800.0 PL=0
MOVL C01094 V=800.0 PL=0
MOVL C01095 V=800.0 PL=0
MOVL C01096 V=800.0 PL=0
MOVL C01097 V=800.0 PL=0
MOVL C01098 V=800.0 PL=0
MOVL C01099 V=800.0 PL=0
MOVL C01100 V=800.0 PL=0
MOVL C01101 V=800.0 PL=0
MOVL C01102 V=800.0 PL=0
MOVL C01103 V=800.0 PL=0
MOVL C01104 V=800.0 PL=0
MOVL C01105 V=800.0 PL=0
MOVL C01106 V=800.0 PL=0
MOVL C01107 V=800.0 PL=0
MOVL C01108 V=800.0 PL=0
MOVL C01109 V=800.0 PL=0
MOVL C01110 V=800.0 PL=0
MOVL C01111 V=800.0 PL=0
MOVL C01112 V=800.0 PL=0
MOVL C01113 V=800.0 PL=0
MOVL C01114 V=800.0 PL=0
MOVL C01115 V=800.0 PL=0
MOVL C01116 V=800.0 PL=0
MOVL C01117 V=800.0 PL=0
MOVL C01118 V=800.0 PL=0
MOVL C01119 V=800.0 PL=0
MOVL C01120 V=800.0 PL=0
MOVL C01121 V=800.0 PL=0
MOVL C01122 V=800.0 PL=0
MOVL C01123 V=800.0 PL=0
MOVL C01124 V=800.0 PL=0
MOVL C01125 V=800.0 PL=0
MOVL C01126 V=800.0 PL=0
MOVL C01127 V=800.0 PL=0
MOVL C01128 V=800.0 PL=0
MOVL C01129 V=800.0 PL=0
MOVL C01130 V=800.0 PL=0
MOVL C01131 V=800.0 PL=0
MOVL C01132 V=800.0 PL=0
MOVL C01133 V=800.0 PL=0
MOVL C01134 V=800.0 PL=0
MOVL C01135 V=800.0 PL=0
MOVL C01136 V=800.0 PL=0
MOVL C01137 V=800.0 PL=0
MOVL C01138 V=800.0 PL=0
MOVL C01139 V=800.0 PL=0
MOVL C01140 V=800.0 PL=0
MOVL C01141 V=800.0 PL=0
MOVL C01142 V=800.0 PL=0
MOVL C01143 V=800.0 PL=0
MOVL C01144 V=800.0 PL=0
MOVL C01145 V=800.0 PL=0
MOVL C01146 V=800.0 PL=0
MOVL C01147 V=800.0 PL=0
MOVL C01148 V=800.0 PL=0
MOVL C01149 V=800.0 PL=0
MOVL C01150 V=800.0 PL=0
MOVL C01151 V=800.0 PL=0
MOVL C01152 V=800.0 PL=0
MOVL C01153 V=800.0 PL=0
MOVL C01154 V=800.0 PL=0
MOVL C01155 V=800.0 PL=0
MOVL C01156 V=800.0 PL=0
MOVL C01157 V=800.0 PL=0
MOVL C01158 V=800.0 PL=0
MOVL C01159 V=800.0 PL=0
MOVL C01160 V=800.0 PL=0
MOVL C01161 V=800.0 PL=0
MOVL C01162 V=800.0 PL=0
MOVL C01163 V=800.0 PL=0
MOVL C01164 V=800.0 PL=0
MOVL C01165 V=800.0 PL=0
MOVL C01166 V=800.0 PL=0
MOVL C01167 V=800.0 PL=0
MOVL C01168 V=800.0 PL=0
MOVL C01169 V=800.0 PL=0
MOVL C01170 V=800.0 PL=0
MOVL C01171 V=800.0 PL=0
MOVL C01172 V=800.0 PL=0
MOVL C01173 V=800.0 PL=0
MOVL C01174 V=800.0 PL=0
MOVL C01175 V=800.0 PL=0
MOVL C01176 V=800.0 PL=0
MOVL C01177 V=800.0 PL=0
MOVL C01178 V=800.0 PL=0
MOVL C01179 V=800.0 PL=0
MOVL C01180 V=800.0 PL=0
MOVL C01181 V=800.0 PL=0
MOVL C01182 V=800.0 PL=0
MOVL C01183 V=800.0 PL=0
MOVL C01184 V=800.0 PL=0
MOVL C01185 V=800.0 PL=0
MOVL C01186 V=800.0 PL=0
MOVL C01187 V=800.0 PL=0
MOVL C01188 V=800.0 PL=0
MOVL C01189 V=800.0 PL=0
MOVL C01190 V=800.0 PL=0
MOVL C01191 V=800.0 PL=0
MOVL C01192 V=800.0 PL=0
MOVL C01193 V=800.0 PL=0
MOVL C01194 V=800.0 PL=0
MOVL C01195 V=800.0 PL=0
MOVL C01196 V=800.0 PL=0
MOVL C01197 V=800.0 PL=0
MOVL C01198 V=800.0 PL=0
MOVL C01199 V=800.0 PL=0
MOVL C01200 V=800.0 PL=0
MOVL C01201 V=800.0 PL=0
MOVL C01202 V=800.0 PL=0
MOVL C01203 V=800.0 PL=0
MOVL C01204 V=800.0 PL=0
MOVL C01205 V=800.0 PL=0
MOVL C01206 V=800.0 PL=0
MOVL C01207 V=800.0 PL=0
MOVL C01208 V=800.0 PL=0
MOVL C01209 V=800.0 PL=0
MOVL C01210 V=800.0 PL=0
MOVL C01211 V=800.0 PL=0
MOVL C01212 V=800.0 PL=0
MOVL C01213 V=800.0 PL=0
MOVL C01214 V=800.0 PL=0
MOVL C01215 V=800.0 PL=0
MOVL C01216 V=800.0 PL=0
MOVL C01217 V=800.0 PL=0
MOVL C01218 V=800.0 PL=0
MOVL C01219 V=800.0 PL=0
MOVL C01220 V=800.0 PL=0
MOVL C01221 V=800.0 PL=0
MOVL C01222 V=800.0 PL=0
MOVL C01223 V=800.0 PL=0
MOVL C01224 V=800.0 PL=0
MOVL C01225 V=800.0 PL=0
MOVL C01226 V=800.0 PL=0
MOVL C01227 V=800.0 PL=0
MOVL C01228 V=800.0 PL=0
MOVL C01229 V=800.0 PL=0
MOVL C01230 V=800.0 PL=0
MOVL C01231 V=800.0 PL=0
MOVL C01232 V=800.0 PL=0
MOVL C01233 V=800.0 PL=0
MOVL C01234 V=800.0 PL=0
MOVL C01235 V=800.0 PL=0
MOVL C01236 V=800.0 PL=0
MOVL C01237 V=800.0 PL=0
MOVL C01238 V=800.0 PL=0
MOVL C01239 V=800.0 PL=0
MOVL C01240 V=800.0 PL=0
MOVL C01241 V=800.0 PL=0
MOVL C01242 V=800.0 PL=0
MOVL C01243 V=800.0 PL=0
MOVL C01244 V=800.0 PL=0
MOVL C01245 V=800.0 PL=0
MOVL C01246 V=800.0 PL=0
MOVL C01247 V=800.0 PL=0
MOVL C01248 V=800.0 PL=0
MOVL C01249 V=800.0 PL=0
MOVL C01250 V=800.0 PL=0
MOVL C01251 V=800.0 PL=0
MOVL C01252 V=800.0 PL=0
MOVL C01253 V=800.0 PL=0
MOVL C01254 V=800.0 PL=0
MOVL C01255 V=800.0 PL=0
MOVL C01256 V=800.0 PL=0
MOVL C01257 V=800.0 PL=0
MOVL C01258 V=800.0 PL=0
MOVL C01259 V=800.0 PL=0
MOVL C01260 V=800.0 PL=0
MOVL C01261 V=800.0 PL=0
MOVL C01262 V=800.0 PL=0
MOVL C01263 V=800.0 PL=0
MOVL C01264 V=800.0 PL=0
MOVL C01265 V=800.0 PL=0
MOVL C01266 V=800.0 PL=0
MOVL C01267 V=800.0 PL=0
MOVL C01268 V=800.0 PL=0
MOVL C01269 V=800.0 PL=0
MOVL C01270 V=800.0 PL=0
MOVL C01271 V=800.0 PL=0
MOVL C01272 V=800.0 PL=0
MOVL C01273 V=800.0 PL=0
MOVL C01274 V=800.0 PL=0
MOVL C01275 V=800.0 PL=0
MOVL C01276 V=800.0 PL=0
MOVL C01277 V=800.0 PL=0
MOVL C01278 V=800.0 PL=0
MOVL C01279 V=800.0 PL=0
MOVL C01280 V=800.0 PL=0
MOVL C01281 V=800.0 PL=0
MOVL C01282 V=800.0 PL=0
MOVL C01283 V=800.0 PL=0
MOVL C01284 V=800.0 PL=0
MOVL C01285 V=800.0 PL=0
MOVL C01286 V=800.0 PL=0
MOVL C01287 V=800.0 PL=0
MOVL C01288 V=800.0 PL=0
MOVL C01289 V=800.0 PL=0
MOVL C01290 V=800.0 PL=0
MOVL C01291 V=800.0 PL=0
MOVL C01292 V=800.0 PL=0
MOVL C01293 V=800.0 PL=0
MOVL C01294 V=800.0 PL=0
MOVL C01295 V=800.0 PL=0
MOVL C01296 V=800.0 PL=0
MOVL C01297 V=800.0 PL=0
MOVL C01298 V=800.0 PL=0
MOVL C01299 V=800.0 PL=0
MOVL C01300 V=800.0 PL=0
MOVL C01301 V=800.0 PL=0
MOVL C01302 V=800.0 PL=0
MOVL C01303 V=800.0 PL=0
MOVL C01304 V=800.0 PL=0
MOVL C01305 V=800.0 PL=0
MOVL C01306 V=800.0 PL=0
MOVL C01307 V=800.0 PL=0
MOVL C01308 V=800.0 PL=0
MOVL C01309 V=800.0 PL=0
MOVL C01310 V=800.0 PL=0
MOVL C01311 V=800.0 PL=0
MOVL C01312 V=800.0 PL=0
MOVL C01313 V=800.0 PL=0
MOVL C01314 V=800.0 PL=0
MOVL C01315 V=800.0 PL=0
MOVL C01316 V=800.0 PL=0
MOVL C01317 V=800.0 PL=0
MOVL C01318 V=800.0 PL=0
MOVL C01319 V=800.0 PL=0
MOVL C01320 V=800.0 PL=0
MOVL C01321 V=800.0 PL=0
MOVL C01322 V=800.0 PL=0
MOVL C01323 V=800.0 PL=0
MOVL C01324 V=800.0 PL=0
MOVL C01325 V=800.0 PL=0
MOVL C01326 V=800.0 PL=0
MOVL C01327 V=800.0 PL=0
MOVL C01328 V=800.0 PL=0
MOVL C01329 V=800.0 PL=0
MOVL C01330 V=800.0 PL=0
MOVL C01331 V=800.0 PL=0
MOVL C01332 V=800.0 PL=0
MOVL C01333 V=800.0 PL=0
MOVL C01334 V=800.0 PL=0
MOVL C01335 V=800.0 PL=0
MOVL C01336 V=800.0 PL=0
MOVL C01337 V=800.0 PL=0
MOVL C01338 V=800.0 PL=0
MOVL C01339 V=800.0 PL=0
MOVL C01340 V=800.0 PL=0
MOVL C01341 V=800.0 PL=0
MOVL C01342 V=800.0 PL=0
MOVL C01343 V=800.0 PL=0
MOVL C01344 V=800.0 PL=0
MOVL C01345 V=800.0 PL=0
MOVL C01346 V=800.0 PL=0
MOVL C01347 V=800.0 PL=0
MOVL C01348 V=800.0 PL=0
MOVL C01349 V=800.0 PL=0
MOVL C01350 V=800.0 PL=0
MOVL C01351 V=800.0 PL=0
MOVL C01352 V=800.0 PL=0
MOVL C01353 V=800.0 PL=0
MOVL C01354 V=800.0 PL=0
MOVL C01355 V=800.0 PL=0
MOVL C01356 V=800.0 PL=0
MOVL C01357 V=800.0 PL=0
MOVL C01358 V=800.0 PL=0
MOVL C01359 V=800.0 PL=0
MOVL C01360 V=800.0 PL=0
MOVL C01361 V=800.0 PL=0
MOVL C01362 V=800.0 PL=0
MOVL C01363 V=800.0 PL=0
MOVL C01364 V=800.0 PL=0
MOVL C01365 V=800.0 PL=0
MOVL C01366 V=800.0 PL=0
MOVL C01367 V=800.0 PL=0
MOVL C01368 V=800.0 PL=0
MOVL C01369 V=800.0 PL=0
MOVL C01370 V=800.0 PL=0
MOVL C01371 V=800.0 PL=0
MOVL C01372 V=800.0 PL=0
MOVL C01373 V=800.0 PL=0
MOVL C01374 V=800.0 PL=0
MOVL C01375 V=800.0 PL=0
MOVL C01376 V=800.0 PL=0
MOVL C01377 V=800.0 PL=0
MOVL C01378 V=800.0 PL=0
MOVL C01379 V=800.0 PL=0
MOVL C01380 V=800.0 PL=0
MOVL C01381 V=800.0 PL=0
MOVL C01382 V=800.0 PL=0
MOVL C01383 V=800.0 PL=0
MOVL C01384 V=800.0 PL=0
MOVL C01385 V=800.0 PL=0
MOVL C01386 V=800.0 PL=0
MOVL C01387 V=800.0 PL=0
MOVL C01388 V=800.0 PL=0
MOVL C01389 V=800.0 PL=0
MOVL C01390 V=800.0 PL=0
MOVL C01391 V=800.0 PL=0
MOVL C01392 V=800.0 PL=0
MOVL C01393 V=800.0 PL=0
MOVL C01394 V=800.0 PL=0
MOVL C01395 V=800.0 PL=0
MOVL C01396 V=800.0 PL=0
MOVL C01397 V=800.0 PL=0
MOVL C01398 V=800.0 PL=0
MOVL C01399 V=800.0 PL=0
MOVL C01400 V=800.0 PL=0
MOVL C01401 V=800.0 PL=0
MOVL C01402 V=800.0 PL=0
MOVL C01403 V=800.0 PL=0
MOVL C01404 V=800.0 PL=0
MOVL C01405 V=800.0 PL=0
MOVL C01406 V=800.0 PL=0
MOVL C01407 V=800.0 PL=0
MOVL C01408 V=800.0 PL=0
MOVL C01409 V=800.0 PL=0
MOVL C01410 V=800.0 PL=0
MOVL C01411 V=800.0 PL=0
MOVL C01412 V=800.0 PL=0
MOVL C01413 V=800.0 PL=0
MOVL C01414 V=800.0 PL=0
MOVL C01415 V=800.0 PL=0
MOVL C01416 V=800.0 PL=0
MOVL C01417 V=800.0 PL=0
MOVL C01418 V=800.0 PL=0
MOVL C01419 V=800.0 PL=0
MOVL C01420 V=800.0 PL=0
MOVL C01421 V=800.0 PL=0
MOVL C01422 V=800.0 PL=0
MOVL C01423 V=800.0 PL=0
MOVL C01424 V=800.0 PL=0
MOVL C01425 V=800.0 PL=0
MOVL C01426 V=800.0 PL=0
MOVL C01427 V=800.0 PL=0
MOVL C01428 V=800.0 PL=0
MOVL C01429 V=800.0 PL=0
MOVL C01430 V=800.0 PL=0
MOVL C01431 V=800.0 PL=0
MOVL C01432 V=800.0 PL=0
MOVL C01433 V=800.0 PL=0
MOVL C01434 V=800.0 PL=0
MOVL C01435 V=800.0 PL=0
MOVL C01436 V=800.0 PL=0
MOVL C01437 V=800.0 PL=0
MOVL C01438 V=800.0 PL=0
MOVL C01439 V=800.0 PL=0
MOVL C01440 V=800.0 PL=0
MOVL C01441 V=800.0 PL=0
MOVL C01442 V=800.0 PL=0
MOVL C01443 V=800.0 PL=0
MOVL C01444 V=800.0 PL=0
MOVL C01445 V=800.0 PL=0
MOVL C01446 V=800.0 PL=0
MOVL C01447 V=800.0 PL=0
MOVL C01448 V=800.0 PL=0
MOVL C01449 V=800.0 PL=0
MOVL C01450 V=800.0 PL=0
MOVL C01451 V=800.0 PL=0
MOVL C01452 V=800.0 PL=0
MOVL C01453 V=800.0 PL=0
MOVL C01454 V=800.0 PL=0
MOVL C01455 V=800.0 PL=0
MOVL C01456 V=800.0 PL=0
MOVL C01457 V=800.0 PL=0
MOVL C01458 V=800.0 PL=0
MOVL C01459 V=800.0 PL=0
MOVL C01460 V=800.0 PL=0
MOVL C01461 V=800.0 PL=0
MOVL C01462 V=800.0 PL=0
MOVL C01463 V=800.0 PL=0
MOVL C01464 V=800.0 PL=0
MOVL C01465 V=800.0 PL=0
MOVL C01466 V=800.0 PL=0
MOVL C01467 V=800.0 PL=0
MOVL C01468 V=800.0 PL=0
MOVL C01469 V=800.0 PL=0
MOVL C01470 V=800.0 PL=0
MOVL C01471 V=800.0 PL=0
MOVL C01472 V=800.0 PL=0
MOVL C01473 V=800.0 PL=0
MOVL C01474 V=800.0 PL=0
MOVL C01475 V=800.0 PL=0
MOVL C01476 V=800.0 PL=0
MOVL C01477 V=800.0 PL=0
MOVL C01478 V=800.0 PL=0
MOVL C01479 V=800.0 PL=0
MOVL C01480 V=800.0 PL=0
MOVL C01481 V=800.0 PL=0
MOVL C01482 V=800.0 PL=0
MOVL C01483 V=800.0 PL=0
MOVL C01484 V=800.0 PL=0
MOVL C01485 V=800.0 PL=0
MOVL C01486 V=800.0 PL=0
MOVL C01487 V=800.0 PL=0
MOVL C01488 V=800.0 PL=0
MOVL C01489 V=800.0 PL=0
MOVL C01490 V=800.0 PL=0
MOVL C01491 V=800.0 PL=0
MOVL C01492 V=800.0 PL=0
MOVL C01493 V=800.0 PL=0
MOVL C01494 V=800.0 PL=0
MOVL C01495 V=800.0 PL=0
MOVL C01496 V=800.0 PL=0
MOVL C01497 V=800.0 PL=0
MOVL C01498 V=800.0 PL=0
MOVL C01499 V=800.0 PL=0
MOVL C01500 V=800.0 PL=0
MOVL C01501 V=800.0 PL=0
MOVL C01502 V=800.0 PL=0
MOVL C01503 V=800.0 PL=0
MOVL C01504 V=800.0 PL=0
MOVL C01505 V=800.0 PL=0
MOVL C01506 V=800.0 PL=0
MOVL C01507 V=800.0 PL=0
MOVL C01508 V=800.0 PL=0
MOVL C01509 V=800.0 PL=0
MOVL C01510 V=800.0 PL=0
MOVL C01511 V=800.0 PL=0
MOVL C01512 V=800.0 PL=0
MOVL C01513 V=800.0 PL=0
MOVL C01514 V=800.0 PL=0
MOVL C01515 V=800.0 PL=0
MOVL C01516 V=800.0 PL=0
MOVL C01517 V=800.0 PL=0
MOVL C01518 V=800.0 PL=0
MOVL C01519 V=800.0 PL=0
MOVL C01520 V=800.0 PL=0
MOVL C01521 V=800.0 PL=0
MOVL C01522 V=800.0 PL=0
MOVL C01523 V=800.0 PL=0
MOVL C01524 V=800.0 PL=0
MOVL C01525 V=800.0 PL=0
MOVL C01526 V=800.0 PL=0
MOVL C01527 V=800.0 PL=0
MOVL C01528 V=800.0 PL=0
MOVL C01529 V=800.0 PL=0
MOVL C01530 V=800.0 PL=0
MOVL C01531 V=800.0 PL=0
MOVL C01532 V=800.0 PL=0
MOVL C01533 V=800.0 PL=0
MOVL C01534 V=800.0 PL=0
MOVL C01535 V=800.0 PL=0
MOVL C01536 V=800.0 PL=0
MOVL C01537 V=800.0 PL=0
MOVL C01538 V=800.0 PL=0
MOVL C01539 V=800.0 PL=0
MOVL C01540 V=800.0 PL=0
MOVL C01541 V=800.0 PL=0
MOVL C01542 V=800.0 PL=0
MOVL C01543 V=800.0 PL=0
MOVL C01544 V=800.0 PL=0
MOVL C01545 V=800.0 PL=0
MOVL C01546 V=800.0 PL=0
MOVL C01547 V=800.0 PL=0
MOVL C01548 V=800.0 PL=0
MOVL C01549 V=800.0 PL=0
MOVL C01550 V=800.0 PL=0
MOVL C01551 V=800.0 PL=0
MOVL C01552 V=800.0 PL=0
MOVL C01553 V=800.0 PL=0
MOVL C01554 V=800.0 PL=0
MOVL C01555 V=800.0 PL=0
MOVL C01556 V=800.0 PL=0
MOVL C01557 V=800.0 PL=0
MOVL C01558 V=800.0 PL=0
MOVL C01559 V=800.0 PL=0
MOVL C01560 V=800.0 PL=0
MOVL C01561 V=800.0 PL=0
MOVL C01562 V=800.0 PL=0
MOVL C01563 V=800.0 PL=0
MOVL C01564 V=800.0 PL=0
MOVL C01565 V=800.0 PL=0
MOVL C01566 V=800.0 PL=0
MOVL C01567 V=800.0 PL=0
MOVL C01568 V=800.0 PL=0
MOVL C01569 V=800.0 PL=0
MOVL C01570 V=800.0 PL=0
MOVL C01571 V=800.0 PL=0
MOVL C01572 V=800.0 PL=0
MOVL C01573 V=800.0 PL=0
MOVL C01574 V=800.0 PL=0
MOVL C01575 V=800.0 PL=0
MOVL C01576 V=800.0 PL=0
MOVL C01577 V=800.0 PL=0
MOVL C01578 V=800.0 PL=0
MOVL C01579 V=800.0 PL=0
MOVL C01580 V=800.0 PL=0
MOVL C01581 V=800.0 PL=0
MOVL C01582 V=800.0 PL=0
MOVL C01583 V=800.0 PL=0
MOVL C01584 V=800.0 PL=0
MOVL C01585 V=800.0 PL=0
MOVL C01586 V=800.0 PL=0
MOVL C01587 V=800.0 PL=0
MOVL C01588 V=800.0 PL=0
MOVL C01589 V=800.0 PL=0
MOVL C01590 V=800.0 PL=0
MOVL C01591 V=800.0 PL=0
MOVL C01592 V=800.0 PL=0
MOVL C01593 V=800.0 PL=0
MOVL C01594 V=800.0 PL=0
MOVL C01595 V=800.0 PL=0
MOVL C01596 V=800.0 PL=0
MOVL C01597 V=800.0 PL=0
MOVL C01598 V=800.0 PL=0
MOVL C01599 V=800.0 PL=0
MOVL C01600 V=800.0 PL=0
MOVL C01601 V=800.0 PL=0
MOVL C01602 V=800.0 PL=0
MOVL C01603 V=800.0 PL=0
MOVL C01604 V=800.0 PL=0
MOVL C01605 V=800.0 PL=0
MOVL C01606 V=800.0 PL=0
MOVL C01607 V=800.0 PL=0
MOVL C01608 V=800.0 PL=0
MOVL C01609 V=800.0 PL=0
MOVL C01610 V=800.0 PL=0
MOVL C01611 V=800.0 PL=0
MOVL C01612 V=800.0 PL=0
MOVL C01613 V=800.0 PL=0
MOVL C01614 V=800.0 PL=0
MOVL C01615 V=800.0 PL=0
MOVL C01616 V=800.0 PL=0
MOVL C01617 V=800.0 PL=0
MOVL C01618 V=800.0 PL=0
MOVL C01619 V=800.0 PL=0
MOVL C01620 V=800.0 PL=0
MOVL C01621 V=800.0 PL=0
MOVL C01622 V=800.0 PL=0
MOVL C01623 V=800.0 PL=0
MOVL C01624 V=800.0 PL=0
MOVL C01625 V=800.0 PL=0
MOVL C01626 V=800.0 PL=0
MOVL C01627 V=800.0 PL=0
MOVL C01628 V=800.0 PL=0
MOVL C01629 V=800.0 PL=0
MOVL C01630 V=800.0 PL=0
MOVL C01631 V=800.0 PL=0
MOVL C01632 V=800.0 PL=0
MOVL C01633 V=800.0 PL=0
MOVL C01634 V=800.0 PL=0
MOVL C01635 V=800.0 PL=0
MOVL C01636 V=800.0 PL=0
MOVL C01637 V=800.0 PL=0
MOVL C01638 V=800.0 PL=0
MOVL C01639 V=800.0 PL=0
MOVL C01640 V=800.0 PL=0
MOVL C01641 V=800.0 PL=0
MOVL C01642 V=800.0 PL=0
MOVL C01643 V=800.0 PL=0
MOVL C01644 V=800.0 PL=0
MOVL C01645 V=800.0 PL=0
MOVL C01646 V=800.0 PL=0
MOVL C01647 V=800.0 PL=0
MOVL C01648 V=800.0 PL=0
MOVL C01649 V=800.0 PL=0
MOVL C01650 V=800.0 PL=0
MOVL C01651 V=800.0 PL=0
MOVL C01652 V=800.0 PL=0
MOVL C01653 V=800.0 PL=0
MOVL C01654 V=800.0 PL=0
MOVL C01655 V=800.0 PL=0
MOVL C01656 V=800.0 PL=0
MOVL C01657 V=800.0 PL=0
MOVL C01658 V=800.0 PL=0
MOVL C01659 V=800.0 PL=0
MOVL C01660 V=800.0 PL=0
MOVL C01661 V=800.0 PL=0
MOVL C01662 V=800.0 PL=0
MOVL C01663 V=800.0 PL=0
MOVL C01664 V=800.0 PL=0
MOVL C01665 V=800.0 PL=0
MOVL C01666 V=800.0 PL=0
MOVL C01667 V=800.0 PL=0
MOVL C01668 V=800.0 PL=0
MOVL C01669 V=800.0 PL=0
MOVL C01670 V=800.0 PL=0
MOVL C01671 V=800.0 PL=0
MOVL C01672 V=800.0 PL=0
MOVL C01673 V=800.0 PL=0
MOVL C01674 V=800.0 PL=0
MOVL C01675 V=800.0 PL=0
MOVL C01676 V=800.0 PL=0
MOVL C01677 V=800.0 PL=0
MOVL C01678 V=800.0 PL=0
MOVL C01679 V=800.0 PL=0
MOVL C01680 V=800.0 PL=0
MOVL C01681 V=800.0 PL=0
MOVL C01682 V=800.0 PL=0
MOVL C01683 V=800.0 PL=0
MOVL C01684 V=800.0 PL=0
MOVL C01685 V=800.0 PL=0
MOVL C01686 V=800.0 PL=0
MOVL C01687 V=800.0 PL=0
MOVL C01688 V=800.0 PL=0
MOVL C01689 V=800.0 PL=0
MOVL C01690 V=800.0 PL=0
MOVL C01691 V=800.0 PL=0
MOVL C01692 V=800.0 PL=0
MOVL C01693 V=800.0 PL=0
MOVL C01694 V=800.0 PL=0
MOVL C01695 V=800.0 PL=0
MOVL C01696 V=800.0 PL=0
MOVL C01697 V=800.0 PL=0
MOVL C01698 V=800.0 PL=0
MOVL C01699 V=800.0 PL=0
MOVL C01700 V=800.0 PL=0
MOVL C01701 V=800.0 PL=0
MOVL C01702 V=800.0 PL=0
MOVL C01703 V=800.0 PL=0
MOVL C01704 V=800.0 PL=0
MOVL C01705 V=800.0 PL=0
MOVL C01706 V=800.0 PL=0
MOVL C01707 V=800.0 PL=0
MOVL C01708 V=800.0 PL=0
MOVL C01709 V=800.0 PL=0
MOVL C01710 V=800.0 PL=0
MOVL C01711 V=800.0 PL=0
MOVL C01712 V=800.0 PL=0
MOVL C01713 V=800.0 PL=0
MOVL C01714 V=800.0 PL=0
MOVL C01715 V=800.0 PL=0
MOVL C01716 V=800.0 PL=0
MOVL C01717 V=800.0 PL=0
MOVL C01718 V=800.0 PL=0
MOVL C01719 V=800.0 PL=0
MOVL C01720 V=800.0 PL=0
MOVL C01721 V=800.0 PL=0
MOVL C01722 V=800.0 PL=0
MOVL C01723 V=800.0 PL=0
MOVL C01724 V=800.0 PL=0
MOVL C01725 V=800.0 PL=0
MOVL C01726 V=800.0 PL=0
MOVL C01727 V=800.0 PL=0
MOVL C01728 V=800.0 PL=0
MOVL C01729 V=800.0 PL=0
MOVL C01730 V=800.0 PL=0
MOVL C01731 V=800.0 PL=0
MOVL C01732 V=800.0 PL=0
MOVL C01733 V=800.0 PL=0
MOVL C01734 V=800.0 PL=0
MOVL C01735 V=800.0 PL=0
MOVL C01736 V=800.0 PL=0
MOVL C01737 V=800.0 PL=0
MOVL C01738 V=800.0 PL=0
MOVL C01739 V=800.0 PL=0
MOVL C01740 V=800.0 PL=0
MOVL C01741 V=800.0 PL=0
MOVL C01742 V=800.0 PL=0
MOVL C01743 V=800.0 PL=0
MOVL C01744 V=800.0 PL=0
MOVL C01745 V=800.0 PL=0
MOVL C01746 V=800.0 PL=0
MOVL C01747 V=800.0 PL=0
MOVL C01748 V=800.0 PL=0
MOVL C01749 V=800.0 PL=0
MOVL C01750 V=800.0 PL=0
MOVL C01751 V=800.0 PL=0
MOVL C01752 V=800.0 PL=0
MOVL C01753 V=800.0 PL=0
MOVL C01754 V=800.0 PL=0
MOVL C01755 V=800.0 PL=0
MOVL C01756 V=800.0 PL=0
MOVL C01757 V=800.0 PL=0
MOVL C01758 V=800.0 PL=0
MOVL C01759 V=800.0 PL=0
MOVL C01760 V=800.0 PL=0
MOVL C01761 V=800.0 PL=0
MOVL C01762 V=800.0 PL=0
MOVL C01763 V=800.0 PL=0
MOVL C01764 V=800.0 PL=0
MOVL C01765 V=800.0 PL=0
MOVL C01766 V=800.0 PL=0
MOVL C01767 V=800.0 PL=0
MOVL C01768 V=800.0 PL=0
MOVL C01769 V=800.0 PL=0
MOVL C01770 V=800.0 PL=0
MOVL C01771 V=800.0 PL=0
MOVL C01772 V=800.0 PL=0
MOVL C01773 V=800.0 PL=0
MOVL C01774 V=800.0 PL=0
MOVL C01775 V=800.0 PL=0
MOVL C01776 V=800.0 PL=0
MOVL C01777 V=800.0 PL=0
MOVL C01778 V=800.0 PL=0
MOVL C01779 V=800.0 PL=0
MOVL C01780 V=800.0 PL=0
MOVL C01781 V=800.0 PL=0
MOVL C01782 V=800.0 PL=0
MOVL C01783 V=800.0 PL=0
MOVL C01784 V=800.0 PL=0
MOVL C01785 V=800.0 PL=0
MOVL C01786 V=800.0 PL=0
MOVL C01787 V=800.0 PL=0
MOVL C01788 V=800.0 PL=0
MOVL C01789 V=800.0 PL=0
MOVL C01790 V=800.0 PL=0
MOVL C01791 V=800.0 PL=0
MOVL C01792 V=800.0 PL=0
MOVL C01793 V=800.0 PL=0
MOVL C01794 V=800.0 PL=0
MOVL C01795 V=800.0 PL=0
MOVL C01796 V=800.0 PL=0
MOVL C01797 V=800.0 PL=0
MOVL C01798 V=800.0 PL=0
MOVL C01799 V=800.0 PL=0
MOVL C01800 V=800.0 PL=0
MOVL C01801 V=800.0 PL=0
MOVL C01802 V=800.0 PL=0
MOVL C01803 V=800.0 PL=0
MOVL C01804 V=800.0 PL=0
MOVL C01805 V=800.0 PL=0
MOVL C01806 V=800.0 PL=0
MOVL C01807 V=800.0 PL=0
MOVL C01808 V=800.0 PL=0
MOVL C01809 V=800.0 PL=0
MOVL C01810 V=800.0 PL=0
MOVL C01811 V=800.0 PL=0
MOVL C01812 V=800.0 PL=0
MOVL C01813 V=800.0 PL=0
MOVL C01814 V=800.0 PL=0
MOVL C01815 V=800.0 PL=0
MOVL C01816 V=800.0 PL=0
MOVL C01817 V=800.0 PL=0
MOVL C01818 V=800.0 PL=0
MOVL C01819 V=800.0 PL=0
MOVL C01820 V=800.0 PL=0
MOVL C01821 V=800.0 PL=0
MOVL C01822 V=800.0 PL=0
MOVL C01823 V=800.0 PL=0
MOVL C01824 V=800.0 PL=0
MOVL C01825 V=800.0 PL=0
MOVL C01826 V=800.0 PL=0
MOVL C01827 V=800.0 PL=0
MOVL C01828 V=800.0 PL=0
MOVL C01829 V=800.0 PL=0
MOVL C01830 V=800.0 PL=0
MOVL C01831 V=800.0 PL=0
MOVL C01832 V=800.0 PL=0
MOVL C01833 V=800.0 PL=0
MOVL C01834 V=800.0 PL=0
MOVL C01835 V=800.0 PL=0
MOVL C01836 V=800.0 PL=0
MOVL C01837 V=800.0 PL=0
MOVL C01838 V=800.0 PL=0
MOVL C01839 V=800.0 PL=0
MOVL C01840 V=800.0 PL=0
MOVL C01841 V=800.0 PL=0
MOVL C01842 V=800.0 PL=0
MOVL C01843 V=800.0 PL=0
MOVL C01844 V=800.0 PL=0
MOVL C01845 V=800.0 PL=0
MOVL C01846 V=800.0 PL=0
MOVL C01847 V=800.0 PL=0
MOVL C01848 V=800.0 PL=0
MOVL C01849 V=800.0 PL=0
MOVL C01850 V=800.0 PL=0
MOVL C01851 V=800.0 PL=0
MOVL C01852 V=800.0 PL=0
MOVL C01853 V=800.0 PL=0
MOVL C01854 V=800.0 PL=0
MOVL C01855 V=800.0 PL=0
MOVL C01856 V=800.0 PL=0
MOVL C01857 V=800.0 PL=0
MOVL C01858 V=800.0 PL=0
MOVL C01859 V=800.0 PL=0
MOVL C01860 V=800.0 PL=0
MOVL C01861 V=800.0 PL=0
MOVL C01862 V=800.0 PL=0
MOVL C01863 V=800.0 PL=0
MOVL C01864 V=800.0 PL=0
MOVL C01865 V=800.0 PL=0
MOVL C01866 V=800.0 PL=0
MOVL C01867 V=800.0 PL=0
MOVL C01868 V=800.0 PL=0
MOVL C01869 V=800.0 PL=0
MOVL C01870 V=800.0 PL=0
MOVL C01871 V=800.0 PL=0
MOVL C01872 V=800.0 PL=0
MOVL C01873 V=800.0 PL=0
MOVL C01874 V=800.0 PL=0
MOVL C01875 V=800.0 PL=0
MOVL C01876 V=800.0 PL=0
MOVL C01877 V=800.0 PL=0
MOVL C01878 V=800.0 PL=0
MOVL C01879 V=800.0 PL=0
MOVL C01880 V=800.0 PL=0
MOVL C01881 V=800.0 PL=0
MOVL C01882 V=800.0 PL=0
MOVL C01883 V=800.0 PL=0
MOVL C01884 V=800.0 PL=0
MOVL C01885 V=800.0 PL=0
MOVL C01886 V=800.0 PL=0
MOVL C01887 V=800.0 PL=0
MOVL C01888 V=800.0 PL=0
MOVL C01889 V=800.0 PL=0
MOVL C01890 V=800.0 PL=0
MOVL C01891 V=800.0 PL=0
MOVL C01892 V=800.0 PL=0
MOVL C01893 V=800.0 PL=0
MOVL C01894 V=800.0 PL=0
MOVL C01895 V=800.0 PL=0
MOVL C01896 V=800.0 PL=0
MOVL C01897 V=800.0 PL=0
MOVL C01898 V=800.0 PL=0
MOVL C01899 V=800.0 PL=0
MOVL C01900 V=800.0 PL=0
MOVL C01901 V=800.0 PL=0
MOVL C01902 V=800.0 PL=0
MOVL C01903 V=800.0 PL=0
MOVL C01904 V=800.0 PL=0
MOVL C01905 V=800.0 PL=0
MOVL C01906 V=800.0 PL=0
MOVL C01907 V=800.0 PL=0
MOVL C01908 V=800.0 PL=0
MOVL C01909 V=800.0 PL=0
MOVL C01910 V=800.0 PL=0
MOVL C01911 V=800.0 PL=0
MOVL C01912 V=800.0 PL=0
MOVL C01913 V=800.0 PL=0
MOVL C01914 V=800.0 PL=0
MOVL C01915 V=800.0 PL=0
MOVL C01916 V=800.0 PL=0
MOVL C01917 V=800.0 PL=0
MOVL C01918 V=800.0 PL=0
MOVL C01919 V=800.0 PL=0
MOVL C01920 V=800.0 PL=0
MOVL C01921 V=800.0 PL=0
MOVL C01922 V=800.0 PL=0
MOVL C01923 V=800.0 PL=0
MOVL C01924 V=800.0 PL=0
MOVL C01925 V=800.0 PL=0
MOVL C01926 V=800.0 PL=0
MOVL C01927 V=800.0 PL=0
MOVL C01928 V=800.0 PL=0
MOVL C01929 V=800.0 PL=0
MOVL C01930 V=800.0 PL=0
MOVL C01931 V=800.0 PL=0
MOVL C01932 V=800.0 PL=0
MOVL C01933 V=800.0 PL=0
MOVL C01934 V=800.0 PL=0
MOVL C01935 V=800.0 PL=0
MOVL C01936 V=800.0 PL=0
MOVL C01937 V=800.0 PL=0
MOVL C01938 V=800.0 PL=0
MOVL C01939 V=800.0 PL=0
MOVL C01940 V=800.0 PL=0
MOVL C01941 V=800.0 PL=0
MOVL C01942 V=800.0 PL=0
MOVL C01943 V=800.0 PL=0
MOVL C01944 V=800.0 PL=0
MOVL C01945 V=800.0 PL=0
MOVL C01946 V=800.0 PL=0
MOVL C01947 V=800.0 PL=0
MOVL C01948 V=800.0 PL=0
MOVL C01949 V=800.0 PL=0
MOVL C01950 V=800.0 PL=0
MOVL C01951 V=800.0 PL=0
MOVL C01952 V=800.0 PL=0
MOVL C01953 V=800.0 PL=0
MOVL C01954 V=800.0 PL=0
MOVL C01955 V=800.0 PL=0
MOVL C01956 V=800.0 PL=0
MOVL C01957 V=800.0 PL=0
MOVL C01958 V=800.0 PL=0
MOVL C01959 V=800.0 PL=0
MOVL C01960 V=800.0 PL=0
MOVL C01961 V=800.0 PL=0
MOVL C01962 V=800.0 PL=0
MOVL C01963 V=800.0 PL=0
MOVL C01964 V=800.0 PL=0
MOVL C01965 V=800.0 PL=0
MOVL C01966 V=800.0 PL=0
MOVL C01967 V=800.0 PL=0
MOVL C01968 V=800.0 PL=0
MOVL C01969 V=800.0 PL=0
MOVL C01970 V=800.0 PL=0
MOVL C01971 V=800.0 PL=0
MOVL C01972 V=800.0 PL=0
MOVL C01973 V=800.0 PL=0
MOVL C01974 V=800.0 PL=0
MOVL C01975 V=800.0 PL=0
MOVL C01976 V=800.0 PL=0
MOVL C01977 V=800.0 PL=0
MOVL C01978 V=800.0 PL=0
MOVL C01979 V=800.0 PL=0
MOVL C01980 V=800.0 PL=0
MOVL C01981 V=800.0 PL=0
MOVL C01982 V=800.0 PL=0
MOVL C01983 V=800.0 PL=0
MOVL C01984 V=800.0 PL=0
MOVL C01985 V=800.0 PL=0
MOVL C01986 V=800.0 PL=0
MOVL C01987 V=800.0 PL=0
MOVL C01988 V=800.0 PL=0
MOVL C01989 V=800.0 PL=0
MOVL C01990 V=800.0 PL=0
MOVL C01991 V=800.0 PL=0
MOVL C01992 V=800.0 PL=0
MOVL C01993 V=800.0 PL=0
MOVL C01994 V=800.0 PL=0
MOVL C01995 V=800.0 PL=0
MOVL C01996 V=800.0 PL=0
MOVL C01997 V=800.0 PL=0
MOVL C01998 V=800.0 PL=0
MOVL C01999 V=800.0 PL=0
MOVL C02000 V=800.0 PL=0
MOVL C02001 V=800.0 PL=0
MOVL C02002 V=800.0 PL=0
MOVL C02003 V=800.0 PL=0
MOVL C02004 V=800.0 PL=0
MOVL C02005 V=800.0 PL=0
MOVL C02006 V=800.0 PL=0
MOVL C02007 V=800.0 PL=0
MOVL C02008 V=800.0 PL=0
MOVL C02009 V=800.0 PL=0
MOVL C02010 V=800.0 PL=0
MOVL C02011 V=800.0 PL=0
MOVL C02012 V=800.0 PL=0
MOVL C02013 V=800.0 PL=0
MOVL C02014 V=800.0 PL=0
MOVL C02015 V=800.0 PL=0
MOVL C02016 V=800.0 PL=0
MOVL C02017 V=800.0 PL=0
MOVL C02018 V=800.0 PL=0
MOVL C02019 V=800.0 PL=0
MOVL C02020 V=800.0 PL=0
MOVL C02021 V=800.0 PL=0
MOVL C02022 V=800.0 PL=0
MOVL C02023 V=800.0 PL=0
MOVL C02024 V=800.0 PL=0
MOVL C02025 V=800.0 PL=0
MOVL C02026 V=800.0 PL=0
MOVL C02027 V=800.0 PL=0
MOVL C02028 V=800.0 PL=0
MOVL C02029 V=800.0 PL=0
MOVL C02030 V=800.0 PL=0
MOVL C02031 V=800.0 PL=0
MOVL C02032 V=800.0 PL=0
MOVL C02033 V=800.0 PL=0
MOVL C02034 V=800.0 PL=0
MOVL C02035 V=800.0 PL=0
MOVL C02036 V=800.0 PL=0
MOVL C02037 V=800.0 PL=0
MOVL C02038 V=800.0 PL=0
MOVL C02039 V=800.0 PL=0
MOVL C02040 V=800.0 PL=0
MOVL C02041 V=800.0 PL=0
MOVL C02042 V=800.0 PL=0
MOVL C02043 V=800.0 PL=0
MOVL C02044 V=800.0 PL=0
MOVL C02045 V=800.0 PL=0
MOVL C02046 V=800.0 PL=0
MOVL C02047 V=800.0 PL=0
MOVL C02048 V=800.0 PL=0
MOVL C02049 V=800.0 PL=0
MOVL C02050 V=800.0 PL=0
MOVL C02051 V=800.0 PL=0
MOVL C02052 V=800.0 PL=0
MOVL C02053 V=800.0 PL=0
MOVL C02054 V=800.0 PL=0
MOVL C02055 V=800.0 PL=0
MOVL C02056 V=800.0 PL=0
MOVL C02057 V=800.0 PL=0
MOVL C02058 V=800.0 PL=0
MOVL C02059 V=800.0 PL=0
MOVL C02060 V=800.0 PL=0
MOVL C02061 V=800.0 PL=0
MOVL C02062 V=800.0 PL=0
MOVL C02063 V=800.0 PL=0
MOVL C02064 V=800.0 PL=0
MOVL C02065 V=800.0 PL=0
MOVL C02066 V=800.0 PL=0
MOVL C02067 V=800.0 PL=0
MOVL C02068 V=800.0 PL=0
MOVL C02069 V=800.0 PL=0
MOVL C02070 V=800.0 PL=0
MOVL C02071 V=800.0 PL=0
MOVL C02072 V=800.0 PL=0
MOVL C02073 V=800.0 PL=0
MOVL C02074 V=800.0 PL=0
MOVL C02075 V=800.0 PL=0
MOVL C02076 V=800.0 PL=0
MOVL C02077 V=800.0 PL=0
MOVL C02078 V=800.0 PL=0
MOVL C02079 V=800.0 PL=0
MOVL C02080 V=800.0 PL=0
MOVL C02081 V=800.0 PL=0
MOVL C02082 V=800.0 PL=0
MOVL C02083 V=800.0 PL=0
MOVL C02084 V=800.0 PL=0
MOVL C02085 V=800.0 PL=0
MOVL C02086 V=800.0 PL=0
MOVL C02087 V=800.0 PL=0
MOVL C02088 V=800.0 PL=0
MOVL C02089 V=800.0 PL=0
MOVL C02090 V=800.0 PL=0
MOVL C02091 V=800.0 PL=0
MOVL C02092 V=800.0 PL=0
MOVL C02093 V=800.0 PL=0
MOVL C02094 V=800.0 PL=0
MOVL C02095 V=800.0 PL=0
MOVL C02096 V=800.0 PL=0
MOVL C02097 V=800.0 PL=0
MOVL C02098 V=800.0 PL=0
MOVL C02099 V=800.0 PL=0
MOVL C02100 V=800.0 PL=0
MOVL C02101 V=800.0 PL=0
MOVL C02102 V=800.0 PL=0
MOVL C02103 V=800.0 PL=0
MOVL C02104 V=800.0 PL=0
MOVL C02105 V=800.0 PL=0
MOVL C02106 V=800.0 PL=0
MOVL C02107 V=800.0 PL=0
MOVL C02108 V=800.0 PL=0
MOVL C02109 V=800.0 PL=0
MOVL C02110 V=800.0 PL=0
MOVL C02111 V=800.0 PL=0
MOVL C02112 V=800.0 PL=0
MOVL C02113 V=800.0 PL=0
MOVL C02114 V=800.0 PL=0
MOVL C02115 V=800.0 PL=0
MOVL C02116 V=800.0 PL=0
MOVL C02117 V=800.0 PL=0
MOVL C02118 V=800.0 PL=0
MOVL C02119 V=800.0 PL=0
MOVL C02120 V=800.0 PL=0
MOVL C02121 V=800.0 PL=0
MOVL C02122 V=800.0 PL=0
MOVL C02123 V=800.0 PL=0
MOVL C02124 V=800.0 PL=0
MOVL C02125 V=800.0 PL=0
MOVL C02126 V=800.0 PL=0
MOVL C02127 V=800.0 PL=0
MOVL C02128 V=800.0 PL=0
MOVL C02129 V=800.0 PL=0
MOVL C02130 V=800.0 PL=0
MOVL C02131 V=800.0 PL=0
MOVL C02132 V=800.0 PL=0
MOVL C02133 V=800.0 PL=0
MOVL C02134 V=800.0 PL=0
MOVL C02135 V=800.0 PL=0
MOVL C02136 V=800.0 PL=0
MOVL C02137 V=800.0 PL=0
MOVL C02138 V=800.0 PL=0
